   LIN {X 7.485, Y -24.478, Z 79.900}
   LaserEnd_Ext()
   LIN {X 6.429, Y -25.478, Z 79.900}
   LaserStart_Ext()
   LIN {X -3.413, Y -25.478, Z 79.900}
   LaserEnd_Ext()
   LIN {X -1.645, Y -26.478, Z 79.900}
   LaserStart_Ext()
   LIN {X 4.818, Y -26.478, Z 79.900}
   LaserEnd_Ext()
   LIN {X 0.768, Y -14.331, Z 80.750}
   LaserStart_Ext()
   LIN {X 0.932, Y -14.309, Z 80.750} C_DIS
   LIN {X 2.973, Y -14.407, Z 80.750} C_DIS
   LIN {X 4.364, Y -15.140, Z 80.750} C_DIS
   LIN {X 4.854, Y -15.396, Z 80.750} C_DIS
   LIN {X 5.246, Y -15.948, Z 80.750} C_DIS
   LIN {X 6.320, Y -17.473, Z 80.750} C_DIS
   LIN {X 6.562, Y -19.321, Z 80.750} C_DIS
   LIN {X 6.608, Y -19.665, Z 80.750} C_DIS
   LIN {X 6.497, Y -19.988, Z 80.750} C_DIS
   LIN {X 5.824, Y -21.931, Z 80.750} C_DIS
   LIN {X 4.592, Y -23.184, Z 80.750} C_DIS
   LIN {X 4.366, Y -23.413, Z 80.750} C_DIS
   LIN {X 3.828, Y -23.616, Z 80.750} C_DIS
   LIN {X 2.307, Y -24.195, Z 80.750} C_DIS
   LIN {X 1.339, Y -24.139, Z 80.750} C_DIS
   LIN {X 0.262, Y -24.074, Z 80.750} C_DIS
   LIN {X -1.038, Y -23.395, Z 80.750} C_DIS
   LIN {X -1.571, Y -23.119, Z 80.750} C_DIS
   LIN {X -1.885, Y -22.728, Z 80.750} C_DIS
   LIN {X -2.870, Y -21.491, Z 80.750} C_DIS
   LIN {X -3.249, Y -19.979, Z 80.750} C_DIS
   LIN {X -3.379, Y -19.468, Z 80.750} C_DIS
   LIN {X -3.052, Y -18.224, Z 80.750} C_DIS
   LIN {X -2.630, Y -16.631, Z 80.750} C_DIS
   LIN {X -2.228, Y -16.209, Z 80.750} C_DIS
   LIN {X -1.186, Y -15.114, Z 80.750} C_DIS
   LIN {X 0.768, Y -14.331, Z 80.750}
   LaserEnd_Ext()
   LIN {X -7.773, Y 38.728, Z 80.750}
   LaserStart_Ext()
   LIN {X -7.349, Y 37.718, Z 80.750} C_DIS
   LIN {X -6.620, Y 35.844, Z 80.750} C_DIS
   LIN {X -6.489, Y 35.509, Z 80.750} C_DIS
   LIN {X -6.365, Y 35.156, Z 80.750} C_DIS
   LIN {X -5.531, Y 32.760, Z 80.750} C_DIS
   LIN {X -5.439, Y 32.415, Z 80.750} C_DIS
   LIN {X -3.813, Y 26.595, Z 80.750} C_DIS
   LIN {X -3.780, Y 26.392, Z 80.750} C_DIS
   LIN {X -2.579, Y 19.576, Z 80.750} C_DIS
   LIN {X -1.969, Y 10.570, Z 80.750} C_DIS
   LIN {X -1.949, Y 8.966, Z 80.750} C_DIS
   LIN {X -2.076, Y 7.182, Z 80.750} C_DIS
   LIN {X -2.401, Y 1.921, Z 80.750} C_DIS
   LIN {X -2.488, Y 1.019, Z 80.750} C_DIS
   LIN {X -2.607, Y 0.242, Z 80.750} C_DIS
   LIN {X -2.989, Y -1.897, Z 80.750} C_DIS
   LIN {X -3.631, Y -5.562, Z 80.750} C_DIS
   LIN {X -4.628, Y -9.518, Z 80.750} C_DIS
   LIN {X -4.693, Y -9.777, Z 80.750} C_DIS
   LIN {X -4.739, Y -9.925, Z 80.750} C_DIS
   LIN {X -5.557, Y -12.604, Z 80.750} C_DIS
   LIN {X -6.774, Y -16.008, Z 80.750} C_DIS
   LIN {X -7.394, Y -19.162, Z 80.750} C_DIS
   LIN {X -6.873, Y -21.827, Z 80.750} C_DIS
   LIN {X -6.688, Y -22.804, Z 80.750} C_DIS
   LIN {X -6.215, Y -23.560, Z 80.750} C_DIS
   LIN {X -5.131, Y -25.266, Z 80.750} C_DIS
   LIN {X -3.475, Y -26.590, Z 80.750} C_DIS
   LIN {X -2.810, Y -27.127, Z 80.750} C_DIS
   LIN {X -0.160, Y -27.846, Z 80.750} C_DIS
   LIN {X 1.444, Y -28.255, Z 80.750} C_DIS
   LIN {X 2.595, Y -28.009, Z 80.750} C_DIS
   LIN {X 5.063, Y -27.544, Z 80.750} C_DIS
   LIN {X 6.110, Y -26.894, Z 80.750} C_DIS
   LIN {X 7.710, Y -25.848, Z 80.750} C_DIS
   LIN {X 8.986, Y -24.226, Z 80.750} C_DIS
   LIN {X 9.540, Y -23.493, Z 80.750} C_DIS
   LIN {X 9.721, Y -22.905, Z 80.750} C_DIS
   LIN {X 10.582, Y -20.217, Z 80.750} C_DIS
   LIN {X 10.827, Y -17.804, Z 80.750} C_DIS
   LIN {X 10.907, Y -16.970, Z 80.750} C_DIS
   LIN {X 10.952, Y -16.292, Z 80.750} C_DIS
   LIN {X 11.122, Y -14.017, Z 80.750} C_DIS
   LIN {X 11.251, Y -11.038, Z 80.750} C_DIS
   LIN {X 11.281, Y -10.215, Z 80.750} C_DIS
   LIN {X 11.280, Y -8.896, Z 80.750} C_DIS
   LIN {X 11.295, Y -5.428, Z 80.750} C_DIS
   LIN {X 11.137, Y -1.887, Z 80.750} C_DIS
   LIN {X 10.979, Y 1.103, Z 80.750} C_DIS
   LIN {X 10.377, Y 5.431, Z 80.750} C_DIS
   LIN {X 9.497, Y 12.340, Z 80.750} C_DIS
   LIN {X 8.336, Y 17.692, Z 80.750} C_DIS
   LIN {X 7.405, Y 21.631, Z 80.750} C_DIS
   LIN {X 6.860, Y 23.249, Z 80.750} C_DIS
   LIN {X 4.606, Y 30.446, Z 80.750} C_DIS
   LIN {X 3.585, Y 33.112, Z 80.750} C_DIS
   LIN {X 3.490, Y 33.339, Z 80.750} C_DIS
   LIN {X 3.345, Y 33.696, Z 80.750} C_DIS
   LIN {X 3.029, Y 34.443, Z 80.750} C_DIS
   LIN {X 1.716, Y 37.545, Z 80.750} C_DIS
   LIN {X 0.683, Y 39.779, Z 80.750} C_DIS
   LIN {X 0.324, Y 40.550, Z 80.750} C_DIS
   LIN {X 0.053, Y 41.100, Z 80.750} C_DIS
   LIN {X -0.525, Y 42.275, Z 80.750} C_DIS
   LIN {X -1.078, Y 43.355, Z 80.750} C_DIS
   LIN {X -1.313, Y 43.811, Z 80.750} C_DIS
   LIN {X -1.598, Y 44.174, Z 80.750} C_DIS
   LIN {X -2.220, Y 44.969, Z 80.750} C_DIS
   LIN {X -3.185, Y 45.502, Z 80.750} C_DIS
   LIN {X -3.743, Y 45.808, Z 80.750} C_DIS
   LIN {X -4.611, Y 45.864, Z 80.750} C_DIS
   LIN {X -5.484, Y 45.922, Z 80.750} C_DIS
   LIN {X -7.839, Y 44.631, Z 80.750} C_DIS
   LIN {X -8.320, Y 43.767, Z 80.750} C_DIS
   LIN {X -8.665, Y 43.160, Z 80.750} C_DIS
   LIN {X -8.736, Y 42.627, Z 80.750} C_DIS
   LIN {X -8.829, Y 41.756, Z 80.750} C_DIS
   LIN {X -8.594, Y 40.838, Z 80.750} C_DIS
   LIN {X -8.473, Y 40.337, Z 80.750} C_DIS
   LIN {X -8.219, Y 39.759, Z 80.750} C_DIS
   LIN {X -7.970, Y 39.192, Z 80.750} C_DIS
   LIN {X -7.773, Y 38.728, Z 80.750}
   LaserEnd_Ext()
   LIN {X -7.280, Y 40.107, Z 80.750}
   LaserStart_Ext()
   LIN {X -7.280, Y 43.580, Z 80.750}
   LaserEnd_Ext()
   LIN {X -6.280, Y 44.345, Z 80.750}
   LaserStart_Ext()
   LIN {X -6.280, Y 37.728, Z 80.750}
   LaserEnd_Ext()
   LIN {X -6.280, Y -18.671, Z 80.750}
   LaserStart_Ext()
   LIN {X -6.280, Y -19.649, Z 80.750}
   LaserEnd_Ext()
   LIN {X -5.280, Y -23.167, Z 80.750}
   LaserStart_Ext()
   LIN {X -5.280, Y -14.799, Z 80.750}
   LaserEnd_Ext()
   LIN {X -5.280, Y 35.081, Z 80.750}
   LaserStart_Ext()
   LIN {X -5.280, Y 44.894, Z 80.750}
   LaserEnd_Ext()
   LIN {X -4.280, Y 44.841, Z 80.750}
   LaserStart_Ext()
   LIN {X -4.280, Y 31.983, Z 80.750}
   LaserEnd_Ext()
   LIN {X -4.280, Y -11.845, Z 80.750}
   LaserStart_Ext()
   LIN {X -4.280, Y -18.961, Z 80.750}
   LaserEnd_Ext()
   LIN {X -4.280, Y -19.984, Z 80.750}
   LaserStart_Ext()
   LIN {X -4.280, Y -24.667, Z 80.750}
   LaserEnd_Ext()
   LIN {X -3.280, Y -25.466, Z 80.750}
   LaserStart_Ext()
   LIN {X -3.280, Y -22.582, Z 80.750}
   LaserEnd_Ext()
   LIN {X -3.280, Y -15.864, Z 80.750}
   LaserStart_Ext()
   LIN {X -3.280, Y -8.261, Z 80.750}
   LaserEnd_Ext()
   LIN {X -3.280, Y 28.402, Z 80.750}
   LaserStart_Ext()
   LIN {X -3.280, Y 44.412, Z 80.750}
   LaserEnd_Ext()
   LIN {X -2.280, Y 43.423, Z 80.750}
   LaserStart_Ext()
   LIN {X -2.280, Y 23.642, Z 80.750}
   LaserEnd_Ext()
   LIN {X -2.280, Y -3.644, Z 80.750}
   LaserStart_Ext()
   LIN {X -2.280, Y -14.813, Z 80.750}
   LaserEnd_Ext()
   LIN {X -2.280, Y -23.824, Z 80.750}
   LaserStart_Ext()
   LIN {X -2.280, Y -26.234, Z 80.750}
   LaserEnd_Ext()
   LIN {X -1.280, Y -26.506, Z 80.750}
   LaserStart_Ext()
   LIN {X -1.280, Y -24.397, Z 80.750}
   LaserEnd_Ext()
   LIN {X -1.280, Y -14.074, Z 80.750}
   LaserStart_Ext()
   LIN {X -1.280, Y 3.847, Z 80.750}
   LaserEnd_Ext()
   LIN {X -1.280, Y 15.194, Z 80.750}
   LaserStart_Ext()
   LIN {X -1.280, Y 41.544, Z 80.750}
   LaserEnd_Ext()
   LIN {X -0.280, Y 39.477, Z 80.750}
   LaserStart_Ext()
   LIN {X -0.280, Y -13.673, Z 80.750}
   LaserEnd_Ext()
   LIN {X -0.280, Y -24.919, Z 80.750}
   LaserStart_Ext()
   LIN {X -0.280, Y -26.777, Z 80.750}
   LaserEnd_Ext()
   LIN {X 0.720, Y -27.039, Z 80.750}
   LaserStart_Ext()
   LIN {X 0.720, Y -25.103, Z 80.750}
   LaserEnd_Ext()
   LIN {X 0.720, Y -13.312, Z 80.750}
   LaserStart_Ext()
   LIN {X 0.720, Y 37.317, Z 80.750}
   LaserEnd_Ext()
   LIN {X 1.720, Y 34.970, Z 80.750}
   LaserStart_Ext()
   LIN {X 1.720, Y -13.346, Z 80.750}
   LaserEnd_Ext()
   LIN {X 1.720, Y -25.163, Z 80.750}
   LaserStart_Ext()
   LIN {X 1.720, Y -27.173, Z 80.750}
   LaserEnd_Ext()
   LIN {X 2.720, Y -26.968, Z 80.750}
   LaserStart_Ext()
   LIN {X 2.720, Y -25.108, Z 80.750}
   LaserEnd_Ext()
   LIN {X 2.720, Y -13.394, Z 80.750}
   LaserStart_Ext()
   LIN {X 2.720, Y 32.574, Z 80.750}
   LaserEnd_Ext()
   LIN {X 3.720, Y 29.928, Z 80.750}
   LaserStart_Ext()
   LIN {X 3.720, Y -13.670, Z 80.750}
   LaserEnd_Ext()
   LIN {X 3.720, Y -24.727, Z 80.750}
   LaserStart_Ext()
   LIN {X 3.720, Y -26.780, Z 80.750}
   LaserEnd_Ext()
   LIN {X 4.720, Y -26.580, Z 80.750}
   LaserStart_Ext()
   LIN {X 4.720, Y -24.348, Z 80.750}
   LaserEnd_Ext()
   LIN {X 4.720, Y -14.198, Z 80.750}
   LaserStart_Ext()
   LIN {X 4.720, Y 26.736, Z 80.750}
   LaserEnd_Ext()
   LIN {X 5.720, Y 23.544, Z 80.750}
   LaserStart_Ext()
   LIN {X 5.720, Y -14.889, Z 80.750}
   LaserEnd_Ext()
   LIN {X 5.720, Y -23.463, Z 80.750}
   LaserStart_Ext()
   LIN {X 5.720, Y -25.954, Z 80.750}
   LaserEnd_Ext()
   LIN {X 6.720, Y -25.300, Z 80.750}
   LaserStart_Ext()
   LIN {X 6.720, Y -22.372, Z 80.750}
   LaserEnd_Ext()
   LIN {X 6.720, Y -16.305, Z 80.750}
   LaserStart_Ext()
   LIN {X 6.720, Y 20.180, Z 80.750}
   LaserEnd_Ext()
   LIN {X 7.720, Y 15.813, Z 80.750}
   LaserStart_Ext()
   LIN {X 7.720, Y -24.217, Z 80.750}
   LaserEnd_Ext()
   LIN {X 8.720, Y -22.757, Z 80.750}
   LaserStart_Ext()
   LIN {X 8.720, Y 10.522, Z 80.750}
   LaserEnd_Ext()
   LIN {X 9.720, Y 2.896, Z 80.750}
   LaserStart_Ext()
   LIN {X 9.720, Y -18.807, Z 80.750}
   LaserEnd_Ext()
   LIN {X -2.785, Y -21.446, Z 81.600}
   LaserStart_Ext()
   LIN {X -2.815, Y -21.328, Z 81.600} C_DIS
   LIN {X -3.299, Y -19.424, Z 81.600} C_DIS
   LIN {X -2.749, Y -17.335, Z 81.600} C_DIS
   LIN {X -2.557, Y -16.588, Z 81.600} C_DIS
   LIN {X -1.920, Y -15.913, Z 81.600} C_DIS
   LIN {X -1.109, Y -15.060, Z 81.600} C_DIS
   LIN {X -0.319, Y -14.744, Z 81.600} C_DIS
   LIN {X 0.911, Y -14.249, Z 81.600} C_DIS
   LIN {X 2.739, Y -14.334, Z 81.600} C_DIS
   LIN {X 3.041, Y -14.348, Z 81.600} C_DIS
   LIN {X 3.248, Y -14.457, Z 81.600} C_DIS
   LIN {X 4.925, Y -15.333, Z 81.600} C_DIS
   LIN {X 6.267, Y -17.224, Z 81.600} C_DIS
   LIN {X 6.396, Y -17.407, Z 81.600} C_DIS
   LIN {X 6.425, Y -17.629, Z 81.600} C_DIS
   LIN {X 6.689, Y -19.597, Z 81.600} C_DIS
   LIN {X 6.055, Y -21.446, Z 81.600} C_DIS
   LIN {X 5.909, Y -21.868, Z 81.600} C_DIS
   LIN {X 5.509, Y -22.274, Z 81.600} C_DIS
   LIN {X 4.458, Y -23.350, Z 81.600} C_DIS
   LIN {X 3.560, Y -23.696, Z 81.600} C_DIS
   LIN {X 2.399, Y -24.138, Z 81.600} C_DIS
   LIN {X 0.648, Y -24.037, Z 81.600} C_DIS
   LIN {X 0.353, Y -24.021, Z 81.600} C_DIS
   LIN {X 0.161, Y -23.922, Z 81.600} C_DIS
   LIN {X -1.482, Y -23.071, Z 81.600} C_DIS
   LIN {X -2.708, Y -21.542, Z 81.600} C_DIS
   LIN {X -2.785, Y -21.446, Z 81.600}
   LaserEnd_Ext()
   LIN {X -6.716, Y -16.014, Z 81.600}
   LaserStart_Ext()
   LIN {X -6.948, Y -17.246, Z 81.600} C_DIS
   LIN {X -7.315, Y -19.127, Z 81.600} C_DIS
   LIN {X -6.705, Y -22.243, Z 81.600} C_DIS
   LIN {X -6.600, Y -22.768, Z 81.600} C_DIS
   LIN {X -6.439, Y -23.019, Z 81.600} C_DIS
   LIN {X -5.037, Y -25.227, Z 81.600} C_DIS
   LIN {X -3.001, Y -26.854, Z 81.600} C_DIS
   LIN {X -2.712, Y -27.082, Z 81.600} C_DIS
   LIN {X -2.128, Y -27.209, Z 81.600} C_DIS
   LIN {X 1.739, Y -28.194, Z 81.600} C_DIS
   LIN {X 5.106, Y -27.475, Z 81.600} C_DIS
   LIN {X 5.297, Y -27.429, Z 81.600} C_DIS
   LIN {X 5.502, Y -27.300, Z 81.600} C_DIS
   LIN {X 7.745, Y -25.833, Z 81.600} C_DIS
   LIN {X 9.324, Y -23.826, Z 81.600} C_DIS
   LIN {X 9.582, Y -23.509, Z 81.600} C_DIS
   LIN {X 9.852, Y -22.677, Z 81.600} C_DIS
   LIN {X 10.664, Y -20.140, Z 81.600} C_DIS
   LIN {X 10.787, Y -18.934, Z 81.600} C_DIS
   LIN {X 10.982, Y -16.892, Z 81.600} C_DIS
   LIN {X 11.093, Y -15.232, Z 81.600} C_DIS
   LIN {X 11.189, Y -13.939, Z 81.600} C_DIS
   LIN {X 11.263, Y -12.246, Z 81.600} C_DIS
   LIN {X 11.340, Y -10.137, Z 81.600} C_DIS
   LIN {X 11.337, Y -6.755, Z 81.600} C_DIS
   LIN {X 11.343, Y -5.350, Z 81.600} C_DIS
   LIN {X 11.279, Y -3.915, Z 81.600} C_DIS
   LIN {X 11.010, Y 1.198, Z 81.600} C_DIS
   LIN {X 9.980, Y 8.597, Z 81.600} C_DIS
   LIN {X 9.457, Y 12.697, Z 81.600} C_DIS
   LIN {X 8.769, Y 15.872, Z 81.600} C_DIS
   LIN {X 7.400, Y 21.660, Z 81.600} C_DIS
   LIN {X 6.600, Y 24.039, Z 81.600} C_DIS
   LIN {X 4.603, Y 30.414, Z 81.600} C_DIS
   LIN {X 3.699, Y 32.775, Z 81.600} C_DIS
   LIN {X 3.615, Y 32.976, Z 81.600} C_DIS
   LIN {X 3.486, Y 33.292, Z 81.600} C_DIS
   LIN {X 3.353, Y 33.628, Z 81.600} C_DIS
   LIN {X 2.053, Y 36.685, Z 81.600} C_DIS
   LIN {X 1.723, Y 37.465, Z 81.600} C_DIS
   LIN {X 1.463, Y 38.027, Z 81.600} C_DIS
   LIN {X 0.328, Y 40.469, Z 81.600} C_DIS
   LIN {X -0.457, Y 42.060, Z 81.600} C_DIS
   LIN {X -0.509, Y 42.165, Z 81.600} C_DIS
   LIN {X -1.381, Y 43.859, Z 81.600} C_DIS
   LIN {X -2.087, Y 44.757, Z 81.600} C_DIS
   LIN {X -2.291, Y 45.015, Z 81.600} C_DIS
   LIN {X -2.683, Y 45.229, Z 81.600} C_DIS
   LIN {X -3.816, Y 45.851, Z 81.600} C_DIS
   LIN {X -4.788, Y 45.913, Z 81.600} C_DIS
   LIN {X -5.557, Y 45.960, Z 81.600} C_DIS
   LIN {X -7.899, Y 44.674, Z 81.600} C_DIS
   LIN {X -8.103, Y 44.309, Z 81.600} C_DIS
   LIN {X -8.736, Y 43.176, Z 81.600} C_DIS
   LIN {X -8.816, Y 42.344, Z 81.600} C_DIS
   LIN {X -8.886, Y 41.697, Z 81.600} C_DIS
   LIN {X -8.738, Y 41.121, Z 81.600} C_DIS
   LIN {X -8.532, Y 40.369, Z 81.600} C_DIS
   LIN {X -8.269, Y 39.774, Z 81.600} C_DIS
   LIN {X -8.027, Y 39.225, Z 81.600} C_DIS
   LIN {X -7.566, Y 38.137, Z 81.600} C_DIS
   LIN {X -7.403, Y 37.752, Z 81.600} C_DIS
   LIN {X -7.225, Y 37.303, Z 81.600} C_DIS
   LIN {X -6.537, Y 35.545, Z 81.600} C_DIS
   LIN {X -5.613, Y 32.910, Z 81.600} C_DIS
   LIN {X -5.573, Y 32.799, Z 81.600} C_DIS
   LIN {X -3.889, Y 26.817, Z 81.600} C_DIS
   LIN {X -3.656, Y 25.742, Z 81.600} C_DIS
   LIN {X -2.630, Y 19.923, Z 81.600} C_DIS
   LIN {X -1.942, Y 9.757, Z 81.600} C_DIS
   LIN {X -1.913, Y 9.438, Z 81.600} C_DIS
   LIN {X -1.913, Y 9.323, Z 81.600} C_DIS
   LIN {X -2.355, Y 2.148, Z 81.600} C_DIS
   LIN {X -2.481, Y 0.845, Z 81.600} C_DIS
   LIN {X -2.653, Y -0.278, Z 81.600} C_DIS
   LIN {X -3.206, Y -3.370, Z 81.600} C_DIS
   LIN {X -3.577, Y -5.490, Z 81.600} C_DIS
   LIN {X -4.234, Y -8.099, Z 81.600} C_DIS
   LIN {X -4.637, Y -9.740, Z 81.600} C_DIS
   LIN {X -4.984, Y -10.889, Z 81.600} C_DIS
   LIN {X -5.530, Y -12.677, Z 81.600} C_DIS
   LIN {X -6.260, Y -14.720, Z 81.600} C_DIS
   LIN {X -6.716, Y -16.014, Z 81.600}
   LaserEnd_Ext()
   LIN {X 5.112, Y -26.360, Z 81.600}
   LaserStart_Ext()
   LIN {X -1.409, Y -26.360, Z 81.600}
   LaserEnd_Ext()
   LIN {X -3.268, Y -25.360, Z 81.600}
   LaserStart_Ext()
   LIN {X 6.641, Y -25.360, Z 81.600}
   LaserEnd_Ext()
   LIN {X 7.632, Y -24.360, Z 81.600}
   LaserStart_Ext()
   LIN {X 4.617, Y -24.360, Z 81.600}
   LaserEnd_Ext()
   LIN {X -1.168, Y -24.360, Z 81.600}
   LaserStart_Ext()
   LIN {X -4.403, Y -24.360, Z 81.600}
   LaserEnd_Ext()
   LIN {X -5.038, Y -23.360, Z 81.600}
   LaserStart_Ext()
   LIN {X -2.532, Y -23.360, Z 81.600}
   LaserEnd_Ext()
   LIN {X 5.846, Y -23.360, Z 81.600}
   LaserStart_Ext()
   LIN {X 8.418, Y -23.360, Z 81.600}
   LaserEnd_Ext()
   LIN {X 8.903, Y -22.360, Z 81.600}
   LaserStart_Ext()
   LIN {X 6.779, Y -22.360, Z 81.600}
   LaserEnd_Ext()
   LIN {X -3.334, Y -22.360, Z 81.600}
   LaserStart_Ext()
   LIN {X -5.662, Y -22.360, Z 81.600}
   LaserEnd_Ext()
   LIN {X -5.859, Y -21.360, Z 81.600}
   LaserStart_Ext()
   LIN {X -3.838, Y -21.360, Z 81.600}
   LaserEnd_Ext()
   LIN {X 7.142, Y -21.360, Z 81.600}
   LaserStart_Ext()
   LIN {X 9.224, Y -21.360, Z 81.600}
   LaserEnd_Ext()
   LIN {X 9.544, Y -20.360, Z 81.600}
   LaserStart_Ext()
   LIN {X 7.485, Y -20.360, Z 81.600}
   LaserEnd_Ext()
   LIN {X -4.093, Y -20.360, Z 81.600}
   LaserStart_Ext()
   LIN {X -6.055, Y -20.360, Z 81.600}
   LaserEnd_Ext()
   LIN {X -6.250, Y -19.360, Z 81.600}
   LaserStart_Ext()
   LIN {X -4.297, Y -19.360, Z 81.600}
   LaserEnd_Ext()
   LIN {X 7.666, Y -19.360, Z 81.600}
   LaserStart_Ext()
   LIN {X 9.739, Y -19.360, Z 81.600}
   LaserEnd_Ext()
   LIN {X 9.837, Y -18.360, Z 81.600}
   LaserStart_Ext()
   LIN {X 7.532, Y -18.360, Z 81.600}
   LaserEnd_Ext()
   LIN {X -4.053, Y -18.360, Z 81.600}
   LaserStart_Ext()
   LIN {X -6.146, Y -18.360, Z 81.600}
   LaserEnd_Ext()
   LIN {X -5.952, Y -17.360, Z 81.600}
   LaserStart_Ext()
   LIN {X -3.789, Y -17.360, Z 81.600}
   LaserEnd_Ext()
   LIN {X 7.398, Y -17.360, Z 81.600}
   LaserStart_Ext()
   LIN {X 9.933, Y -17.360, Z 81.600}
   LaserEnd_Ext()
   LIN {X 10.015, Y -16.360, Z 81.600}
   LaserStart_Ext()
   LIN {X 6.880, Y -16.360, Z 81.600}
   LaserEnd_Ext()
   LIN {X -3.531, Y -16.360, Z 81.600}
   LaserStart_Ext()
   LIN {X -5.764, Y -16.360, Z 81.600}
   LaserEnd_Ext()
   LIN {X -5.425, Y -15.360, Z 81.600}
   LaserStart_Ext()
   LIN {X -2.773, Y -15.360, Z 81.600}
   LaserEnd_Ext()
   LIN {X 6.170, Y -15.360, Z 81.600}
   LaserStart_Ext()
   LIN {X 10.082, Y -15.360, Z 81.600}
   LaserEnd_Ext()
   LIN {X 10.155, Y -14.360, Z 81.600}
   LaserStart_Ext()
   LIN {X 5.222, Y -14.360, Z 81.600}
   LaserEnd_Ext()
   LIN {X -1.822, Y -14.360, Z 81.600}
   LaserStart_Ext()
   LIN {X -5.070, Y -14.360, Z 81.600}
   LaserEnd_Ext()
   LIN {X -4.712, Y -13.360, Z 81.600}
   LaserStart_Ext()
   LIN {X 0.441, Y -13.360, Z 81.600}
   LaserEnd_Ext()
   LIN {X 3.193, Y -13.360, Z 81.600}
   LaserStart_Ext()
   LIN {X 10.214, Y -13.360, Z 81.600}
   LaserEnd_Ext()
   LIN {X 10.257, Y -12.360, Z 81.600}
   LaserStart_Ext()
   LIN {X -4.388, Y -12.360, Z 81.600}
   LaserEnd_Ext()
   LIN {X -4.082, Y -11.360, Z 81.600}
   LaserStart_Ext()
   LIN {X 10.295, Y -11.360, Z 81.600}
   LaserEnd_Ext()
   LIN {X 10.331, Y -10.360, Z 81.600}
   LaserStart_Ext()
   LIN {X -3.779, Y -10.360, Z 81.600}
   LaserEnd_Ext()
   LIN {X -3.514, Y -9.360, Z 81.600}
   LaserStart_Ext()
   LIN {X 10.339, Y -9.360, Z 81.600}
   LaserEnd_Ext()
   LIN {X 10.338, Y -8.360, Z 81.600}
   LaserStart_Ext()
   LIN {X -3.269, Y -8.360, Z 81.600}
   LaserEnd_Ext()
   LIN {X -3.017, Y -7.360, Z 81.600}
   LaserStart_Ext()
   LIN {X 10.337, Y -7.360, Z 81.600}
   LaserEnd_Ext()
   LIN {X 10.338, Y -6.360, Z 81.600}
   LaserStart_Ext()
   LIN {X -2.765, Y -6.360, Z 81.600}
   LaserEnd_Ext()
   LIN {X -2.539, Y -5.360, Z 81.600}
   LaserStart_Ext()
   LIN {X 10.342, Y -5.360, Z 81.600}
   LaserEnd_Ext()
   LIN {X 10.298, Y -4.360, Z 81.600}
   LaserStart_Ext()
   LIN {X -2.364, Y -4.360, Z 81.600}
   LaserEnd_Ext()
   LIN {X -2.188, Y -3.360, Z 81.600}
   LaserStart_Ext()
   LIN {X 10.248, Y -3.360, Z 81.600}
   LaserEnd_Ext()
   LIN {X 10.196, Y -2.360, Z 81.600}
   LaserStart_Ext()
   LIN {X -2.009, Y -2.360, Z 81.600}
   LaserEnd_Ext()
   LIN {X -1.831, Y -1.360, Z 81.600}
   LaserStart_Ext()
   LIN {X 10.143, Y -1.360, Z 81.600}
   LaserEnd_Ext()
   LIN {X 10.090, Y -0.360, Z 81.600}
   LaserStart_Ext()
   LIN {X -1.654, Y -0.360, Z 81.600}
   LaserEnd_Ext()
   LIN {X -1.501, Y 0.640, Z 81.600}
   LaserStart_Ext()
   LIN {X 10.038, Y 0.640, Z 81.600}
   LaserEnd_Ext()
   LIN {X 9.939, Y 1.640, Z 81.600}
   LaserStart_Ext()
   LIN {X -1.400, Y 1.640, Z 81.600}
   LaserEnd_Ext()
   LIN {X -1.323, Y 2.640, Z 81.600}
   LaserStart_Ext()
   LIN {X 9.800, Y 2.640, Z 81.600}
   LaserEnd_Ext()
   LIN {X 9.660, Y 3.640, Z 81.600}
   LaserStart_Ext()
   LIN {X -1.261, Y 3.640, Z 81.600}
   LaserEnd_Ext()
   LIN {X -1.200, Y 4.640, Z 81.600}
   LaserStart_Ext()
   LIN {X 9.521, Y 4.640, Z 81.600}
   LaserEnd_Ext()
   LIN {X 9.382, Y 5.640, Z 81.600}
   LaserStart_Ext()
   LIN {X -1.138, Y 5.640, Z 81.600}
   LaserEnd_Ext()
   LIN {X -1.076, Y 6.640, Z 81.600}
   LaserStart_Ext()
   LIN {X 9.243, Y 6.640, Z 81.600}
   LaserEnd_Ext()
   LIN {X 9.103, Y 7.640, Z 81.600}
   LaserStart_Ext()
   LIN {X -1.015, Y 7.640, Z 81.600}
   LaserEnd_Ext()
   LIN {X -0.953, Y 8.640, Z 81.600}
   LaserStart_Ext()
   LIN {X 8.966, Y 8.640, Z 81.600}
   LaserEnd_Ext()
   LIN {X 8.839, Y 9.640, Z 81.600}
   LaserStart_Ext()
   LIN {X -0.927, Y 9.640, Z 81.600}
   LaserEnd_Ext()
   LIN {X -1.000, Y 10.640, Z 81.600}
   LaserStart_Ext()
   LIN {X 8.711, Y 10.640, Z 81.600}
   LaserEnd_Ext()
   LIN {X 8.584, Y 11.640, Z 81.600}
   LaserStart_Ext()
   LIN {X -1.067, Y 11.640, Z 81.600}
   LaserEnd_Ext()
   LIN {X -1.135, Y 12.640, Z 81.600}
   LaserStart_Ext()
   LIN {X 8.447, Y 12.640, Z 81.600}
   LaserEnd_Ext()
   LIN {X 8.230, Y 13.640, Z 81.600}
   LaserStart_Ext()
   LIN {X -1.202, Y 13.640, Z 81.600}
   LaserEnd_Ext()
   LIN {X -1.270, Y 14.640, Z 81.600}
   LaserStart_Ext()
   LIN {X 8.013, Y 14.640, Z 81.600}
   LaserEnd_Ext()
   LIN {X 7.796, Y 15.640, Z 81.600}
   LaserStart_Ext()
   LIN {X -1.338, Y 15.640, Z 81.600}
   LaserEnd_Ext()
   LIN {X -1.405, Y 16.640, Z 81.600}
   LaserStart_Ext()
   LIN {X 7.560, Y 16.640, Z 81.600}
   LaserEnd_Ext()
   LIN {X 7.323, Y 17.640, Z 81.600}
   LaserStart_Ext()
   LIN {X -1.473, Y 17.640, Z 81.600}
   LaserEnd_Ext()
   LIN {X -1.541, Y 18.640, Z 81.600}
   LaserStart_Ext()
   LIN {X 7.087, Y 18.640, Z 81.600}
   LaserEnd_Ext()
   LIN {X 6.850, Y 19.640, Z 81.600}
   LaserStart_Ext()
   LIN {X -1.608, Y 19.640, Z 81.600}
   LaserEnd_Ext()
   LIN {X -1.741, Y 20.640, Z 81.600}
   LaserStart_Ext()
   LIN {X 6.614, Y 20.640, Z 81.600}
   LaserEnd_Ext()
   LIN {X 6.352, Y 21.640, Z 81.600}
   LaserStart_Ext()
   LIN {X -1.917, Y 21.640, Z 81.600}
   LaserEnd_Ext()
   LIN {X -2.093, Y 22.640, Z 81.600}
   LaserStart_Ext()
   LIN {X 6.016, Y 22.640, Z 81.600}
   LaserEnd_Ext()
   LIN {X 5.679, Y 23.640, Z 81.600}
   LaserStart_Ext()
   LIN {X -2.270, Y 23.640, Z 81.600}
   LaserEnd_Ext()
   LIN {X -2.446, Y 24.640, Z 81.600}
   LaserStart_Ext()
   LIN {X 5.364, Y 24.640, Z 81.600}
   LaserEnd_Ext()
   LIN {X 5.051, Y 25.640, Z 81.600}
   LaserStart_Ext()
   LIN {X -2.622, Y 25.640, Z 81.600}
   LaserEnd_Ext()
   LIN {X -2.828, Y 26.640, Z 81.600}
   LaserStart_Ext()
   LIN {X 4.738, Y 26.640, Z 81.600}
   LaserEnd_Ext()
   LIN {X 4.424, Y 27.640, Z 81.600}
   LaserStart_Ext()
   LIN {X -3.082, Y 27.640, Z 81.600}
   LaserEnd_Ext()
   LIN {X -3.364, Y 28.640, Z 81.600}
   LaserStart_Ext()
   LIN {X 4.111, Y 28.640, Z 81.600}
   LaserEnd_Ext()
   LIN {X 3.798, Y 29.640, Z 81.600}
   LaserStart_Ext()
   LIN {X -3.645, Y 29.640, Z 81.600}
   LaserEnd_Ext()
   LIN {X -3.926, Y 30.640, Z 81.600}
   LaserStart_Ext()
   LIN {X 3.446, Y 30.640, Z 81.600}
   LaserEnd_Ext()
   LIN {X 3.063, Y 31.640, Z 81.600}
   LaserStart_Ext()
   LIN {X -4.208, Y 31.640, Z 81.600}
   LaserEnd_Ext()
   LIN {X -4.489, Y 32.640, Z 81.600}
   LaserStart_Ext()
   LIN {X 2.672, Y 32.640, Z 81.600}
   LaserEnd_Ext()
   LIN {X 2.261, Y 33.640, Z 81.600}
   LaserStart_Ext()
   LIN {X -4.809, Y 33.640, Z 81.600}
   LaserEnd_Ext()
   LIN {X -5.160, Y 34.640, Z 81.600}
   LaserStart_Ext()
   LIN {X 1.836, Y 34.640, Z 81.600}
   LaserEnd_Ext()
   LIN {X 1.411, Y 35.640, Z 81.600}
   LaserStart_Ext()
   LIN {X -5.511, Y 35.640, Z 81.600}
   LaserEnd_Ext()
   LIN {X -5.892, Y 36.640, Z 81.600}
   LaserStart_Ext()
   LIN {X 0.987, Y 36.640, Z 81.600}
   LaserEnd_Ext()
   LIN {X 0.540, Y 37.640, Z 81.600}
   LaserStart_Ext()
   LIN {X -6.284, Y 37.640, Z 81.600}
   LaserEnd_Ext()
   LIN {X -6.693, Y 38.640, Z 81.600}
   LaserStart_Ext()
   LIN {X 0.076, Y 38.640, Z 81.600}
   LaserEnd_Ext()
   LIN {X -0.389, Y 39.640, Z 81.600}
   LaserStart_Ext()
   LIN {X -7.117, Y 39.640, Z 81.600}
   LaserEnd_Ext()
   LIN {X -7.559, Y 40.640, Z 81.600}
   LaserStart_Ext()
   LIN {X -0.871, Y 40.640, Z 81.600}
   LaserEnd_Ext()
   LIN {X -1.365, Y 41.640, Z 81.600}
   LaserStart_Ext()
   LIN {X -7.839, Y 41.640, Z 81.600}
   LaserEnd_Ext()
   LIN {X -7.783, Y 42.640, Z 81.600}
   LaserStart_Ext()
   LIN {X -1.878, Y 42.640, Z 81.600}
   LaserEnd_Ext()
   LIN {X -2.480, Y 43.640, Z 81.600}
   LaserStart_Ext()
   LIN {X -7.331, Y 43.640, Z 81.600}
   LaserEnd_Ext()
   LIN {X -5.884, Y 44.640, Z 81.600}
   LaserStart_Ext()
   LIN {X -3.688, Y 44.640, Z 81.600}
   LaserEnd_Ext()
   LIN {X -3.044, Y -20.068, Z 82.450}
   LaserStart_Ext()
   LIN {X -3.219, Y -19.380, Z 82.450} C_DIS
   LIN {X -3.042, Y -18.710, Z 82.450} C_DIS
   LIN {X -2.490, Y -16.552, Z 82.450} C_DIS
   LIN {X -1.313, Y -15.306, Z 82.450} C_DIS
   LIN {X -1.047, Y -15.017, Z 82.450} C_DIS
   LIN {X -0.475, Y -14.782, Z 82.450} C_DIS
   LIN {X 0.987, Y -14.194, Z 82.450} C_DIS
   LIN {X 2.062, Y -14.244, Z 82.450} C_DIS
   LIN {X 3.110, Y -14.289, Z 82.450} C_DIS
   LIN {X 4.242, Y -14.876, Z 82.450} C_DIS
   LIN {X 4.995, Y -15.270, Z 82.450} C_DIS
   LIN {X 5.569, Y -16.077, Z 82.450} C_DIS
   LIN {X 6.472, Y -17.340, Z 82.450} C_DIS
   LIN {X 6.647, Y -18.614, Z 82.450} C_DIS
   LIN {X 6.770, Y -19.530, Z 82.450} C_DIS
   LIN {X 6.410, Y -20.579, Z 82.450} C_DIS
   LIN {X 6.012, Y -21.775, Z 82.450} C_DIS
   LIN {X 5.381, Y -22.437, Z 82.450} C_DIS
   LIN {X 4.551, Y -23.285, Z 82.450} C_DIS
   LIN {X 2.592, Y -24.041, Z 82.450} C_DIS
   LIN {X 2.491, Y -24.080, Z 82.450} C_DIS
   LIN {X 0.444, Y -23.969, Z 82.450} C_DIS
   LIN {X -0.955, Y -23.250, Z 82.450} C_DIS
   LIN {X -1.393, Y -23.023, Z 82.450} C_DIS
   LIN {X -1.764, Y -22.561, Z 82.450} C_DIS
   LIN {X -2.700, Y -21.401, Z 82.450} C_DIS
   LIN {X -3.044, Y -20.068, Z 82.450}
   LaserEnd_Ext()
   LIN {X 11.056, Y -16.815, Z 82.450}
   LaserStart_Ext()
   LIN {X 11.234, Y -14.172, Z 82.450} C_DIS
   LIN {X 11.257, Y -13.861, Z 82.450} C_DIS
   LIN {X 11.275, Y -13.454, Z 82.450} C_DIS
   LIN {X 11.399, Y -10.058, Z 82.450} C_DIS
   LIN {X 11.395, Y -5.797, Z 82.450} C_DIS
   LIN {X 11.391, Y -5.271, Z 82.450} C_DIS
   LIN {X 11.376, Y -5.087, Z 82.450} C_DIS
   LIN {X 11.041, Y 1.292, Z 82.450} C_DIS
   LIN {X 9.583, Y 11.764, Z 82.450} C_DIS
   LIN {X 9.418, Y 13.054, Z 82.450} C_DIS
   LIN {X 9.202, Y 14.053, Z 82.450} C_DIS
   LIN {X 7.396, Y 21.690, Z 82.450} C_DIS
   LIN {X 6.340, Y 24.828, Z 82.450} C_DIS
   LIN {X 4.601, Y 30.381, Z 82.450} C_DIS
   LIN {X 3.813, Y 32.438, Z 82.450} C_DIS
   LIN {X 3.740, Y 32.613, Z 82.450} C_DIS
   LIN {X 3.628, Y 32.889, Z 82.450} C_DIS
   LIN {X 3.391, Y 33.487, Z 82.450} C_DIS
   LIN {X 2.033, Y 36.681, Z 82.450} C_DIS
   LIN {X 1.691, Y 37.473, Z 82.450} C_DIS
   LIN {X 0.373, Y 40.302, Z 82.450} C_DIS
   LIN {X 0.265, Y 40.521, Z 82.450} C_DIS
   LIN {X -0.666, Y 42.396, Z 82.450} C_DIS
   LIN {X -1.364, Y 43.746, Z 82.450} C_DIS
   LIN {X -1.449, Y 43.907, Z 82.450} C_DIS
   LIN {X -1.579, Y 44.072, Z 82.450} C_DIS
   LIN {X -2.362, Y 45.060, Z 82.450} C_DIS
   LIN {X -3.513, Y 45.689, Z 82.450} C_DIS
   LIN {X -3.889, Y 45.893, Z 82.450} C_DIS
   LIN {X -4.715, Y 45.942, Z 82.450} C_DIS
   LIN {X -5.630, Y 45.998, Z 82.450} C_DIS
   LIN {X -6.290, Y 45.636, Z 82.450} C_DIS
   LIN {X -7.981, Y 44.692, Z 82.450} C_DIS
   LIN {X -8.592, Y 43.589, Z 82.450} C_DIS
   LIN {X -8.798, Y 43.220, Z 82.450} C_DIS
   LIN {X -8.846, Y 42.721, Z 82.450} C_DIS
   LIN {X -8.949, Y 41.722, Z 82.450} C_DIS
   LIN {X -8.720, Y 40.868, Z 82.450} C_DIS
   LIN {X -8.592, Y 40.400, Z 82.450} C_DIS
   LIN {X -8.374, Y 39.909, Z 82.450} C_DIS
   LIN {X -8.084, Y 39.257, Z 82.450} C_DIS
   LIN {X -7.855, Y 38.723, Z 82.450} C_DIS
   LIN {X -7.456, Y 37.786, Z 82.450} C_DIS
   LIN {X -6.772, Y 36.049, Z 82.450} C_DIS
   LIN {X -6.586, Y 35.581, Z 82.450} C_DIS
   LIN {X -6.429, Y 35.143, Z 82.450} C_DIS
   LIN {X -5.615, Y 32.837, Z 82.450} C_DIS
   LIN {X -5.409, Y 32.177, Z 82.450} C_DIS
   LIN {X -3.977, Y 27.086, Z 82.450} C_DIS
   LIN {X -3.479, Y 24.799, Z 82.450} C_DIS
   LIN {X -2.681, Y 20.270, Z 82.450} C_DIS
   LIN {X -2.146, Y 12.358, Z 82.450} C_DIS
   LIN {X -1.912, Y 9.787, Z 82.450} C_DIS
   LIN {X -1.910, Y 8.861, Z 82.450} C_DIS
   LIN {X -2.310, Y 2.375, Z 82.450} C_DIS
   LIN {X -2.475, Y 0.671, Z 82.450} C_DIS
   LIN {X -2.700, Y -0.798, Z 82.450} C_DIS
   LIN {X -3.422, Y -4.842, Z 82.450} C_DIS
   LIN {X -3.523, Y -5.418, Z 82.450} C_DIS
   LIN {X -3.702, Y -6.126, Z 82.450} C_DIS
   LIN {X -4.571, Y -9.670, Z 82.450} C_DIS
   LIN {X -5.320, Y -12.152, Z 82.450} C_DIS
   LIN {X -5.503, Y -12.750, Z 82.450} C_DIS
   LIN {X -5.746, Y -13.432, Z 82.450} C_DIS
   LIN {X -6.643, Y -15.978, Z 82.450} C_DIS
   LIN {X -7.101, Y -18.403, Z 82.450} C_DIS
   LIN {X -7.235, Y -19.093, Z 82.450} C_DIS
   LIN {X -7.012, Y -20.236, Z 82.450} C_DIS
   LIN {X -6.511, Y -22.732, Z 82.450} C_DIS
   LIN {X -5.748, Y -23.920, Z 82.450} C_DIS
   LIN {X -4.943, Y -25.187, Z 82.450} C_DIS
   LIN {X -3.775, Y -26.121, Z 82.450} C_DIS
   LIN {X -2.613, Y -27.036, Z 82.450} C_DIS
   LIN {X -0.265, Y -27.547, Z 82.450} C_DIS
   LIN {X 2.035, Y -28.133, Z 82.450} C_DIS
   LIN {X 4.036, Y -27.706, Z 82.450} C_DIS
   LIN {X 5.309, Y -27.402, Z 82.450} C_DIS
   LIN {X 6.677, Y -26.540, Z 82.450} C_DIS
   LIN {X 7.780, Y -25.818, Z 82.450} C_DIS
   LIN {X 8.557, Y -24.831, Z 82.450} C_DIS
   LIN {X 9.626, Y -23.515, Z 82.450} C_DIS
   LIN {X 10.747, Y -20.064, Z 82.450} C_DIS
   LIN {X 11.056, Y -16.815, Z 82.450}
   LaserEnd_Ext()
   LIN {X 9.602, Y -20.352, Z 82.450}
   LaserStart_Ext()
   LIN {X 9.602, Y 4.373, Z 82.450}
   LaserEnd_Ext()
   LIN {X 8.602, Y 11.556, Z 82.450}
   LaserStart_Ext()
   LIN {X 8.602, Y -23.190, Z 82.450}
   LaserEnd_Ext()
   LIN {X 7.602, Y -24.428, Z 82.450}
   LaserStart_Ext()
   LIN {X 7.602, Y -20.187, Z 82.450}
   LaserEnd_Ext()
   LIN {X 7.602, Y -18.218, Z 82.450}
   LaserStart_Ext()
   LIN {X 7.602, Y 16.472, Z 82.450}
   LaserEnd_Ext()
   LIN {X 6.602, Y 20.702, Z 82.450}
   LaserStart_Ext()
   LIN {X 6.602, Y -15.803, Z 82.450}
   LaserEnd_Ext()
   LIN {X 6.602, Y -22.605, Z 82.450}
   LaserStart_Ext()
   LIN {X 6.602, Y -25.394, Z 82.450}
   LaserEnd_Ext()
   LIN {X 5.602, Y -26.035, Z 82.450}
   LaserStart_Ext()
   LIN {X 5.602, Y -23.641, Z 82.450}
   LaserEnd_Ext()
   LIN {X 5.602, Y -14.475, Z 82.450}
   LaserStart_Ext()
   LIN {X 5.602, Y 23.887, Z 82.450}
   LaserEnd_Ext()
   LIN {X 4.602, Y 27.033, Z 82.450}
   LaserStart_Ext()
   LIN {X 4.602, Y -13.936, Z 82.450}
   LaserEnd_Ext()
   LIN {X 4.602, Y -24.337, Z 82.450}
   LaserStart_Ext()
   LIN {X 4.602, Y -26.543, Z 82.450}
   LaserEnd_Ext()
   LIN {X 3.602, Y -26.776, Z 82.450}
   LaserStart_Ext()
   LIN {X 3.602, Y -24.723, Z 82.450}
   LaserEnd_Ext()
   LIN {X 3.602, Y -13.418, Z 82.450}
   LaserStart_Ext()
   LIN {X 3.602, Y 30.194, Z 82.450}
   LaserEnd_Ext()
   LIN {X 2.602, Y 32.763, Z 82.450}
   LaserStart_Ext()
   LIN {X 2.602, Y -13.266, Z 82.450}
   LaserEnd_Ext()
   LIN {X 2.602, Y -25.073, Z 82.450}
   LaserStart_Ext()
   LIN {X 2.602, Y -26.990, Z 82.450}
   LaserEnd_Ext()
   LIN {X 1.602, Y -26.991, Z 82.450}
   LaserStart_Ext()
   LIN {X 1.602, Y -25.034, Z 82.450}
   LaserEnd_Ext()
   LIN {X 1.602, Y -13.221, Z 82.450}
   LaserStart_Ext()
   LIN {X 1.602, Y 35.138, Z 82.450}
   LaserEnd_Ext()
   LIN {X 0.602, Y 37.443, Z 82.450}
   LaserStart_Ext()
   LIN {X 0.602, Y -13.271, Z 82.450}
   LaserEnd_Ext()
   LIN {X 0.602, Y -24.979, Z 82.450}
   LaserStart_Ext()
   LIN {X 0.602, Y -26.736, Z 82.450}
   LaserEnd_Ext()
   LIN {X -0.398, Y -26.495, Z 82.450}
   LaserStart_Ext()
   LIN {X -0.398, Y -24.660, Z 82.450}
   LaserEnd_Ext()
   LIN {X -0.398, Y -13.673, Z 82.450}
   LaserStart_Ext()
   LIN {X -0.398, Y 39.588, Z 82.450}
   LaserEnd_Ext()
   LIN {X -1.398, Y 41.623, Z 82.450}
   LaserStart_Ext()
   LIN {X -1.398, Y 16.119, Z 82.450}
   LaserEnd_Ext()
   LIN {X -1.398, Y 1.419, Z 82.450}
   LaserStart_Ext()
   LIN {X -1.398, Y -14.080, Z 82.450}
   LaserEnd_Ext()
   LIN {X -1.398, Y -24.146, Z 82.450}
   LaserStart_Ext()
   LIN {X -1.398, Y -26.277, Z 82.450}
   LaserEnd_Ext()
   LIN {X -2.398, Y -25.933, Z 82.450}
   LaserStart_Ext()
   LIN {X -2.398, Y -23.368, Z 82.450}
   LaserEnd_Ext()
   LIN {X -2.398, Y -14.999, Z 82.450}
   LaserStart_Ext()
   LIN {X -2.398, Y -4.795, Z 82.450}
   LaserEnd_Ext()
   LIN {X -2.398, Y 24.424, Z 82.450}
   LaserStart_Ext()
   LIN {X -2.398, Y 43.495, Z 82.450}
   LaserEnd_Ext()
   LIN {X -3.398, Y 44.487, Z 82.450}
   LaserStart_Ext()
   LIN {X -3.398, Y 28.720, Z 82.450}
   LaserEnd_Ext()
   LIN {X -3.398, Y -9.086, Z 82.450}
   LaserStart_Ext()
   LIN {X -3.398, Y -16.136, Z 82.450}
   LaserEnd_Ext()
   LIN {X -3.398, Y -22.128, Z 82.450}
   LaserStart_Ext()
   LIN {X -3.398, Y -25.142, Z 82.450}
   LaserEnd_Ext()
   LIN {X -4.398, Y -24.180, Z 82.450}
   LaserStart_Ext()
   LIN {X -4.398, Y -12.557, Z 82.450}
   LaserEnd_Ext()
   LIN {X -4.398, Y 32.274, Z 82.450}
   LaserStart_Ext()
   LIN {X -4.398, Y 44.922, Z 82.450}
   LaserEnd_Ext()
   LIN {X -5.398, Y 44.982, Z 82.450}
   LaserStart_Ext()
   LIN {X -5.398, Y 35.225, Z 82.450}
   LaserEnd_Ext()
   LIN {X -5.398, Y -15.453, Z 82.450}
   LaserStart_Ext()
   LIN {X -5.398, Y -22.615, Z 82.450}
   LaserEnd_Ext()
   LIN {X -6.398, Y 37.828, Z 82.450}
   LaserStart_Ext()
   LIN {X -6.398, Y 44.430, Z 82.450}
   LaserEnd_Ext()
   LIN {X -7.398, Y 43.681, Z 82.450}
   LaserStart_Ext()
   LIN {X -7.398, Y 40.175, Z 82.450}
   LaserEnd_Ext()
   LIN {X -3.138, Y -19.336, Z 83.300}
   LaserStart_Ext()
   LIN {X -2.716, Y -17.663, Z 83.300} C_DIS
   LIN {X -2.422, Y -16.516, Z 83.300} C_DIS
   LIN {X -2.110, Y -16.186, Z 83.300} C_DIS
   LIN {X -1.014, Y -14.995, Z 83.300} C_DIS
   LIN {X 0.866, Y -14.222, Z 83.300} C_DIS
   LIN {X 1.063, Y -14.139, Z 83.300} C_DIS
   LIN {X 1.319, Y -14.150, Z 83.300} C_DIS
   LIN {X 3.179, Y -14.230, Z 83.300} C_DIS
   LIN {X 4.531, Y -14.932, Z 83.300} C_DIS
   LIN {X 5.066, Y -15.206, Z 83.300} C_DIS
   LIN {X 5.537, Y -15.860, Z 83.300} C_DIS
   LIN {X 6.548, Y -17.273, Z 83.300} C_DIS
   LIN {X 6.764, Y -18.847, Z 83.300} C_DIS
   LIN {X 6.851, Y -19.462, Z 83.300} C_DIS
   LIN {X 6.661, Y -20.051, Z 83.300} C_DIS
   LIN {X 6.123, Y -21.670, Z 83.300} C_DIS
   LIN {X 4.691, Y -23.171, Z 83.300} C_DIS
   LIN {X 4.607, Y -23.235, Z 83.300} C_DIS
   LIN {X 2.593, Y -24.021, Z 83.300} C_DIS
   LIN {X 1.236, Y -23.954, Z 83.300} C_DIS
   LIN {X 0.536, Y -23.916, Z 83.300} C_DIS
   LIN {X -0.314, Y -23.480, Z 83.300} C_DIS
   LIN {X -1.304, Y -22.974, Z 83.300} C_DIS
   LIN {X -1.840, Y -22.315, Z 83.300} C_DIS
   LIN {X -2.615, Y -21.356, Z 83.300} C_DIS
   LIN {X -2.946, Y -20.071, Z 83.300} C_DIS
   LIN {X -3.138, Y -19.336, Z 83.300}
   LaserEnd_Ext()
   LIN {X -5.703, Y 46.036, Z 83.300}
   LaserStart_Ext()
   LIN {X -7.467, Y 45.040, Z 83.300} C_DIS
   LIN {X -8.069, Y 44.704, Z 83.300} C_DIS
   LIN {X -8.264, Y 44.352, Z 83.300} C_DIS
   LIN {X -8.860, Y 43.265, Z 83.300} C_DIS
   LIN {X -8.989, Y 42.091, Z 83.300} C_DIS
   LIN {X -9.017, Y 41.816, Z 83.300} C_DIS
   LIN {X -8.947, Y 41.554, Z 83.300} C_DIS
   LIN {X -8.652, Y 40.431, Z 83.300} C_DIS
   LIN {X -8.362, Y 39.784, Z 83.300} C_DIS
   LIN {X -8.141, Y 39.289, Z 83.300} C_DIS
   LIN {X -7.721, Y 38.309, Z 83.300} C_DIS
   LIN {X -7.510, Y 37.819, Z 83.300} C_DIS
   LIN {X -7.309, Y 37.317, Z 83.300} C_DIS
   LIN {X -6.634, Y 35.617, Z 83.300} C_DIS
   LIN {X -5.694, Y 32.979, Z 83.300} C_DIS
   LIN {X -5.657, Y 32.875, Z 83.300} C_DIS
   LIN {X -5.252, Y 31.576, Z 83.300} C_DIS
   LIN {X -4.064, Y 27.355, Z 83.300} C_DIS
   LIN {X -3.303, Y 23.856, Z 83.300} C_DIS
   LIN {X -2.732, Y 20.617, Z 83.300} C_DIS
   LIN {X -2.350, Y 14.959, Z 83.300} C_DIS
   LIN {X -1.911, Y 10.136, Z 83.300} C_DIS
   LIN {X -1.908, Y 8.398, Z 83.300} C_DIS
   LIN {X -2.265, Y 2.602, Z 83.300} C_DIS
   LIN {X -2.469, Y 0.497, Z 83.300} C_DIS
   LIN {X -2.746, Y -1.318, Z 83.300} C_DIS
   LIN {X -3.392, Y -4.932, Z 83.300} C_DIS
   LIN {X -3.496, Y -5.473, Z 83.300} C_DIS
   LIN {X -3.789, Y -6.681, Z 83.300} C_DIS
   LIN {X -4.505, Y -9.601, Z 83.300} C_DIS
   LIN {X -5.203, Y -11.913, Z 83.300} C_DIS
   LIN {X -5.440, Y -12.714, Z 83.300} C_DIS
   LIN {X -5.725, Y -13.541, Z 83.300} C_DIS
   LIN {X -6.571, Y -15.942, Z 83.300} C_DIS
   LIN {X -7.033, Y -18.393, Z 83.300} C_DIS
   LIN {X -7.155, Y -19.058, Z 83.300} C_DIS
   LIN {X -7.055, Y -19.542, Z 83.300} C_DIS
   LIN {X -6.423, Y -22.696, Z 83.300} C_DIS
   LIN {X -5.056, Y -24.822, Z 83.300} C_DIS
   LIN {X -4.849, Y -25.147, Z 83.300} C_DIS
   LIN {X -4.549, Y -25.387, Z 83.300} C_DIS
   LIN {X -2.515, Y -26.991, Z 83.300} C_DIS
   LIN {X 1.598, Y -27.886, Z 83.300} C_DIS
   LIN {X 2.330, Y -28.073, Z 83.300} C_DIS
   LIN {X 2.966, Y -27.936, Z 83.300} C_DIS
   LIN {X 5.321, Y -27.375, Z 83.300} C_DIS
   LIN {X 7.789, Y -25.820, Z 83.300} C_DIS
   LIN {X 9.671, Y -23.521, Z 83.300} C_DIS
   LIN {X 10.436, Y -21.165, Z 83.300} C_DIS
   LIN {X 10.830, Y -19.986, Z 83.300} C_DIS
   LIN {X 10.937, Y -18.772, Z 83.300} C_DIS
   LIN {X 11.131, Y -16.737, Z 83.300} C_DIS
   LIN {X 11.272, Y -14.638, Z 83.300} C_DIS
   LIN {X 11.325, Y -13.783, Z 83.300} C_DIS
   LIN {X 11.361, Y -12.639, Z 83.300} C_DIS
   LIN {X 11.458, Y -9.980, Z 83.300} C_DIS
   LIN {X 11.455, Y -7.364, Z 83.300} C_DIS
   LIN {X 11.438, Y -5.193, Z 83.300} C_DIS
   LIN {X 11.377, Y -4.429, Z 83.300} C_DIS
   LIN {X 11.071, Y 1.387, Z 83.300} C_DIS
   LIN {X 9.499, Y 12.677, Z 83.300} C_DIS
   LIN {X 9.422, Y 13.171, Z 83.300} C_DIS
   LIN {X 9.298, Y 13.657, Z 83.300} C_DIS
   LIN {X 7.391, Y 21.720, Z 83.300} C_DIS
   LIN {X 6.080, Y 25.618, Z 83.300} C_DIS
   LIN {X 4.598, Y 30.349, Z 83.300} C_DIS
   LIN {X 3.927, Y 32.101, Z 83.300} C_DIS
   LIN {X 3.865, Y 32.250, Z 83.300} C_DIS
   LIN {X 3.769, Y 32.485, Z 83.300} C_DIS
   LIN {X 3.428, Y 33.345, Z 83.300} C_DIS
   LIN {X 2.495, Y 35.539, Z 83.300} C_DIS
   LIN {X 1.640, Y 37.524, Z 83.300} C_DIS
   LIN {X 0.998, Y 38.903, Z 83.300} C_DIS
   LIN {X 0.338, Y 40.306, Z 83.300} C_DIS
   LIN {X -0.759, Y 42.500, Z 83.300} C_DIS
   LIN {X -0.823, Y 42.627, Z 83.300} C_DIS
   LIN {X -0.870, Y 42.719, Z 83.300} C_DIS
   LIN {X -1.517, Y 43.955, Z 83.300} C_DIS
   LIN {X -2.348, Y 45.000, Z 83.300} C_DIS
   LIN {X -2.432, Y 45.106, Z 83.300} C_DIS
   LIN {X -2.655, Y 45.226, Z 83.300} C_DIS
   LIN {X -3.961, Y 45.935, Z 83.300} C_DIS
   LIN {X -4.774, Y 45.983, Z 83.300} C_DIS
   LIN {X -5.703, Y 46.036, Z 83.300}
   LaserEnd_Ext()
   LIN {X -3.453, Y 44.522, Z 83.300}
   LaserStart_Ext()
   LIN {X -6.351, Y 44.522, Z 83.300}
   LaserEnd_Ext()
   LIN {X -7.579, Y 43.522, Z 83.300}
   LaserStart_Ext()
   LIN {X -2.450, Y 43.522, Z 83.300}
   LaserEnd_Ext()
   LIN {X -1.896, Y 42.522, Z 83.300}
   LaserStart_Ext()
   LIN {X -7.936, Y 42.522, Z 83.300}
   LaserEnd_Ext()
   LIN {X -7.904, Y 41.522, Z 83.300}
   LaserStart_Ext()
   LIN {X -1.388, Y 41.522, Z 83.300}
   LaserEnd_Ext()
   LIN {X -0.888, Y 40.522, Z 83.300}
   LaserStart_Ext()
   LIN {X -7.596, Y 40.522, Z 83.300}
   LaserEnd_Ext()
   LIN {X -7.152, Y 39.522, Z 83.300}
   LaserStart_Ext()
   LIN {X -0.399, Y 39.522, Z 83.300}
   LaserEnd_Ext()
   LIN {X 0.072, Y 38.522, Z 83.300}
   LaserStart_Ext()
   LIN {X -6.723, Y 38.522, Z 83.300}
   LaserEnd_Ext()
   LIN {X -6.314, Y 37.522, Z 83.300}
   LaserStart_Ext()
   LIN {X 0.538, Y 37.522, Z 83.300}
   LaserEnd_Ext()
   LIN {X 0.983, Y 36.522, Z 83.300}
   LaserStart_Ext()
   LIN {X -5.917, Y 36.522, Z 83.300}
   LaserEnd_Ext()
   LIN {X -5.539, Y 35.522, Z 83.300}
   LaserStart_Ext()
   LIN {X 1.414, Y 35.522, Z 83.300}
   LaserEnd_Ext()
   LIN {X 1.841, Y 34.522, Z 83.300}
   LaserStart_Ext()
   LIN {X -5.182, Y 34.522, Z 83.300}
   LaserEnd_Ext()
   LIN {X -4.826, Y 33.522, Z 83.300}
   LaserStart_Ext()
   LIN {X 2.266, Y 33.522, Z 83.300}
   LaserEnd_Ext()
   LIN {X 2.679, Y 32.522, Z 83.300}
   LaserStart_Ext()
   LIN {X -4.500, Y 32.522, Z 83.300}
   LaserEnd_Ext()
   LIN {X -4.198, Y 31.522, Z 83.300}
   LaserStart_Ext()
   LIN {X 3.078, Y 31.522, Z 83.300}
   LaserEnd_Ext()
   LIN {X 3.461, Y 30.522, Z 83.300}
   LaserStart_Ext()
   LIN {X -3.917, Y 30.522, Z 83.300}
   LaserEnd_Ext()
   LIN {X -3.635, Y 29.522, Z 83.300}
   LaserStart_Ext()
   LIN {X 3.810, Y 29.522, Z 83.300}
   LaserEnd_Ext()
   LIN {X 4.123, Y 28.522, Z 83.300}
   LaserStart_Ext()
   LIN {X -3.354, Y 28.522, Z 83.300}
   LaserEnd_Ext()
   LIN {X -3.077, Y 27.522, Z 83.300}
   LaserStart_Ext()
   LIN {X 4.436, Y 27.522, Z 83.300}
   LaserEnd_Ext()
   LIN {X 4.749, Y 26.522, Z 83.300}
   LaserStart_Ext()
   LIN {X -2.860, Y 26.522, Z 83.300}
   LaserEnd_Ext()
   LIN {X -2.642, Y 25.522, Z 83.300}
   LaserStart_Ext()
   LIN {X 5.063, Y 25.522, Z 83.300}
   LaserEnd_Ext()
   LIN {X 5.394, Y 24.522, Z 83.300}
   LaserStart_Ext()
   LIN {X -2.425, Y 24.522, Z 83.300}
   LaserEnd_Ext()
   LIN {X -2.229, Y 23.522, Z 83.300}
   LaserStart_Ext()
   LIN {X 5.730, Y 23.522, Z 83.300}
   LaserEnd_Ext()
   LIN {X 6.067, Y 22.522, Z 83.300}
   LaserStart_Ext()
   LIN {X -2.053, Y 22.522, Z 83.300}
   LaserEnd_Ext()
   LIN {X -1.877, Y 21.522, Z 83.300}
   LaserStart_Ext()
   LIN {X 6.403, Y 21.522, Z 83.300}
   LaserEnd_Ext()
   LIN {X 6.647, Y 20.522, Z 83.300}
   LaserStart_Ext()
   LIN {X -1.724, Y 20.522, Z 83.300}
   LaserEnd_Ext()
   LIN {X -1.656, Y 19.522, Z 83.300}
   LaserStart_Ext()
   LIN {X 6.884, Y 19.522, Z 83.300}
   LaserEnd_Ext()
   LIN {X 7.120, Y 18.522, Z 83.300}
   LaserStart_Ext()
   LIN {X -1.588, Y 18.522, Z 83.300}
   LaserEnd_Ext()
   LIN {X -1.521, Y 17.522, Z 83.300}
   LaserStart_Ext()
   LIN {X 7.356, Y 17.522, Z 83.300}
   LaserEnd_Ext()
   LIN {X 7.593, Y 16.522, Z 83.300}
   LaserStart_Ext()
   LIN {X -1.453, Y 16.522, Z 83.300}
   LaserEnd_Ext()
   LIN {X -1.385, Y 15.522, Z 83.300}
   LaserStart_Ext()
   LIN {X 7.829, Y 15.522, Z 83.300}
   LaserEnd_Ext()
   LIN {X 8.066, Y 14.522, Z 83.300}
   LaserStart_Ext()
   LIN {X -1.306, Y 14.522, Z 83.300}
   LaserEnd_Ext()
   LIN {X -1.215, Y 13.522, Z 83.300}
   LaserStart_Ext()
   LIN {X 8.302, Y 13.522, Z 83.300}
   LaserEnd_Ext()
   LIN {X 8.511, Y 12.522, Z 83.300}
   LaserStart_Ext()
   LIN {X -1.124, Y 12.522, Z 83.300}
   LaserEnd_Ext()
   LIN {X -1.033, Y 11.522, Z 83.300}
   LaserStart_Ext()
   LIN {X 8.650, Y 11.522, Z 83.300}
   LaserEnd_Ext()
   LIN {X 8.790, Y 10.522, Z 83.300}
   LaserStart_Ext()
   LIN {X -0.942, Y 10.522, Z 83.300}
   LaserEnd_Ext()
   LIN {X -0.910, Y 9.522, Z 83.300}
   LaserStart_Ext()
   LIN {X 8.929, Y 9.522, Z 83.300}
   LaserEnd_Ext()
   LIN {X 9.068, Y 8.522, Z 83.300}
   LaserStart_Ext()
   LIN {X -0.908, Y 8.522, Z 83.300}
   LaserEnd_Ext()
   LIN {X -0.960, Y 7.522, Z 83.300}
   LaserStart_Ext()
   LIN {X 9.207, Y 7.522, Z 83.300}
   LaserEnd_Ext()
   LIN {X 9.347, Y 6.522, Z 83.300}
   LaserStart_Ext()
   LIN {X -1.021, Y 6.522, Z 83.300}
   LaserEnd_Ext()
   LIN {X -1.083, Y 5.522, Z 83.300}
   LaserStart_Ext()
   LIN {X 9.486, Y 5.522, Z 83.300}
   LaserEnd_Ext()
   LIN {X 9.625, Y 4.522, Z 83.300}
   LaserStart_Ext()
   LIN {X -1.145, Y 4.522, Z 83.300}
   LaserEnd_Ext()
   LIN {X -1.206, Y 3.522, Z 83.300}
   LaserStart_Ext()
   LIN {X 9.764, Y 3.522, Z 83.300}
   LaserEnd_Ext()
   LIN {X 9.903, Y 2.522, Z 83.300}
   LaserStart_Ext()
   LIN {X -1.268, Y 2.522, Z 83.300}
   LaserEnd_Ext()
   LIN {X -1.365, Y 1.522, Z 83.300}
   LaserStart_Ext()
   LIN {X 10.043, Y 1.522, Z 83.300}
   LaserEnd_Ext()
   LIN {X 10.115, Y 0.522, Z 83.300}
   LaserStart_Ext()
   LIN {X -1.462, Y 0.522, Z 83.300}
   LaserEnd_Ext()
   LIN {X -1.606, Y -0.478, Z 83.300}
   LaserStart_Ext()
   LIN {X 10.168, Y -0.478, Z 83.300}
   LaserEnd_Ext()
   LIN {X 10.220, Y -1.478, Z 83.300}
   LaserStart_Ext()
   LIN {X -1.759, Y -1.478, Z 83.300}
   LaserEnd_Ext()
   LIN {X -1.938, Y -2.478, Z 83.300}
   LaserStart_Ext()
   LIN {X 10.273, Y -2.478, Z 83.300}
   LaserEnd_Ext()
   LIN {X 10.325, Y -3.478, Z 83.300}
   LaserStart_Ext()
   LIN {X -2.116, Y -3.478, Z 83.300}
   LaserEnd_Ext()
   LIN {X -2.295, Y -4.478, Z 83.300}
   LaserStart_Ext()
   LIN {X 10.378, Y -4.478, Z 83.300}
   LaserEnd_Ext()
   LIN {X 10.440, Y -5.478, Z 83.300}
   LaserStart_Ext()
   LIN {X -2.478, Y -5.478, Z 83.300}
   LaserEnd_Ext()
   LIN {X -2.711, Y -6.478, Z 83.300}
   LaserStart_Ext()
   LIN {X 10.448, Y -6.478, Z 83.300}
   LaserEnd_Ext()
   LIN {X 10.455, Y -7.478, Z 83.300}
   LaserStart_Ext()
   LIN {X -2.955, Y -7.478, Z 83.300}
   LaserEnd_Ext()
   LIN {X -3.200, Y -8.478, Z 83.300}
   LaserStart_Ext()
   LIN {X 10.456, Y -8.478, Z 83.300}
   LaserEnd_Ext()
   LIN {X 10.457, Y -9.478, Z 83.300}
   LaserStart_Ext()
   LIN {X -3.446, Y -9.478, Z 83.300}
   LaserEnd_Ext()
   LIN {X -3.726, Y -10.478, Z 83.300}
   LaserStart_Ext()
   LIN {X 10.439, Y -10.478, Z 83.300}
   LaserEnd_Ext()
   LIN {X 10.402, Y -11.478, Z 83.300}
   LaserStart_Ext()
   LIN {X -4.027, Y -11.478, Z 83.300}
   LaserEnd_Ext()
   LIN {X -4.327, Y -12.478, Z 83.300}
   LaserStart_Ext()
   LIN {X 10.366, Y -12.478, Z 83.300}
   LaserEnd_Ext()
   LIN {X 10.334, Y -13.478, Z 83.300}
   LaserStart_Ext()
   LIN {X 3.901, Y -13.478, Z 83.300}
   LaserEnd_Ext()
   LIN {X 0.046, Y -13.478, Z 83.300}
   LaserStart_Ext()
   LIN {X -4.645, Y -13.478, Z 83.300}
   LaserEnd_Ext()
   LIN {X -4.995, Y -14.478, Z 83.300}
   LaserStart_Ext()
   LIN {X -1.898, Y -14.478, Z 83.300}
   LaserEnd_Ext()
   LIN {X 5.752, Y -14.478, Z 83.300}
   LaserStart_Ext()
   LIN {X 10.280, Y -14.478, Z 83.300}
   LaserEnd_Ext()
   LIN {X 10.214, Y -15.478, Z 83.300}
   LaserStart_Ext()
   LIN {X 6.494, Y -15.478, Z 83.300}
   LaserEnd_Ext()
   LIN {X -2.818, Y -15.478, Z 83.300}
   LaserStart_Ext()
   LIN {X -5.347, Y -15.478, Z 83.300}
   LaserEnd_Ext()
   LIN {X -5.654, Y -16.478, Z 83.300}
   LaserStart_Ext()
   LIN {X -3.444, Y -16.478, Z 83.300}
   LaserEnd_Ext()
   LIN {X 7.209, Y -16.478, Z 83.300}
   LaserStart_Ext()
   LIN {X 10.146, Y -16.478, Z 83.300}
   LaserEnd_Ext()
   LIN {X 10.056, Y -17.478, Z 83.300}
   LaserStart_Ext()
   LIN {X 7.585, Y -17.478, Z 83.300}
   LaserEnd_Ext()
   LIN {X -3.700, Y -17.478, Z 83.300}
   LaserStart_Ext()
   LIN {X -5.843, Y -17.478, Z 83.300}
   LaserEnd_Ext()
   LIN {X -6.031, Y -18.478, Z 83.300}
   LaserStart_Ext()
   LIN {X -3.953, Y -18.478, Z 83.300}
   LaserEnd_Ext()
   LIN {X 7.723, Y -18.478, Z 83.300}
   LaserStart_Ext()
   LIN {X 9.961, Y -18.478, Z 83.300}
   LaserEnd_Ext()
   LIN {X 9.871, Y -19.478, Z 83.300}
   LaserStart_Ext()
   LIN {X 7.850, Y -19.478, Z 83.300}
   LaserEnd_Ext()
   LIN {X -4.127, Y -19.478, Z 83.300}
   LaserStart_Ext()
   LIN {X -6.048, Y -19.478, Z 83.300}
   LaserEnd_Ext()
   LIN {X -5.847, Y -20.478, Z 83.300}
   LaserStart_Ext()
   LIN {X -3.874, Y -20.478, Z 83.300}
   LaserEnd_Ext()
   LIN {X 7.573, Y -20.478, Z 83.300}
   LaserStart_Ext()
   LIN {X 9.611, Y -20.478, Z 83.300}
   LaserEnd_Ext()
   LIN {X 9.283, Y -21.478, Z 83.300}
   LaserStart_Ext()
   LIN {X 7.240, Y -21.478, Z 83.300}
   LaserEnd_Ext()
   LIN {X -3.616, Y -21.478, Z 83.300}
   LaserStart_Ext()
   LIN {X -5.647, Y -21.478, Z 83.300}
   LaserEnd_Ext()
   LIN {X -5.374, Y -22.478, Z 83.300}
   LaserStart_Ext()
   LIN {X -2.994, Y -22.478, Z 83.300}
   LaserEnd_Ext()
   LIN {X 6.733, Y -22.478, Z 83.300}
   LaserStart_Ext()
   LIN {X 8.958, Y -22.478, Z 83.300}
   LaserEnd_Ext()
   LIN {X 8.417, Y -23.478, Z 83.300}
   LaserStart_Ext()
   LIN {X 5.780, Y -23.478, Z 83.300}
   LaserEnd_Ext()
   LIN {X -2.183, Y -23.478, Z 83.300}
   LaserStart_Ext()
   LIN {X -4.731, Y -23.478, Z 83.300}
   LaserEnd_Ext()
   LIN {X -4.085, Y -24.478, Z 83.300}
   LaserStart_Ext()
   LIN {X -0.558, Y -24.478, Z 83.300}
   LaserEnd_Ext()
   LIN {X 4.172, Y -24.478, Z 83.300}
   LaserStart_Ext()
   LIN {X 7.605, Y -24.478, Z 83.300}
   LaserEnd_Ext()
   LIN {X 6.455, Y -25.478, Z 83.300}
   LaserStart_Ext()
   LIN {X -2.818, Y -25.478, Z 83.300}
   LaserEnd_Ext()
   LIN {X -0.167, Y -26.478, Z 83.300}
   LaserStart_Ext()
   LIN {X 4.769, Y -26.478, Z 83.300}
   LaserEnd_Ext()
   LIN {X -2.559, Y -21.198, Z 84.150}
   LaserStart_Ext()
   LIN {X -3.058, Y -19.292, Z 84.150} C_DIS
   LIN {X -2.579, Y -17.398, Z 84.150} C_DIS
   LIN {X -2.354, Y -16.480, Z 84.150} C_DIS
   LIN {X -1.630, Y -15.678, Z 84.150} C_DIS
   LIN {X -0.982, Y -14.973, Z 84.150} C_DIS
   LIN {X -0.310, Y -14.697, Z 84.150} C_DIS
   LIN {X 1.140, Y -14.083, Z 84.150} C_DIS
   LIN {X 3.021, Y -14.162, Z 84.150} C_DIS
   LIN {X 3.247, Y -14.172, Z 84.150} C_DIS
   LIN {X 3.412, Y -14.257, Z 84.150} C_DIS
   LIN {X 5.138, Y -15.143, Z 84.150} C_DIS
   LIN {X 6.591, Y -17.162, Z 84.150} C_DIS
   LIN {X 6.631, Y -17.256, Z 84.150} C_DIS
   LIN {X 6.932, Y -19.395, Z 84.150} C_DIS
   LIN {X 6.243, Y -21.534, Z 84.150} C_DIS
   LIN {X 4.736, Y -23.156, Z 84.150} C_DIS
   LIN {X 3.536, Y -23.634, Z 84.150} C_DIS
   LIN {X 2.696, Y -23.962, Z 84.150} C_DIS
   LIN {X 1.432, Y -23.900, Z 84.150} C_DIS
   LIN {X 0.627, Y -23.863, Z 84.150} C_DIS
   LIN {X 0.122, Y -23.608, Z 84.150} C_DIS
   LIN {X -1.215, Y -22.926, Z 84.150} C_DIS
   LIN {X -2.449, Y -21.408, Z 84.150} C_DIS
   LIN {X -2.529, Y -21.310, Z 84.150} C_DIS
   LIN {X -2.559, Y -21.198, Z 84.150}
   LaserEnd_Ext()
   LIN {X -1.905, Y 7.936, Z 84.150}
   LaserStart_Ext()
   LIN {X -2.220, Y 2.830, Z 84.150} C_DIS
   LIN {X -2.462, Y 0.323, Z 84.150} C_DIS
   LIN {X -2.793, Y -1.838, Z 84.150} C_DIS
   LIN {X -3.215, Y -4.200, Z 84.150} C_DIS
   LIN {X -3.484, Y -5.603, Z 84.150} C_DIS
   LIN {X -4.244, Y -8.736, Z 84.150} C_DIS
   LIN {X -4.440, Y -9.531, Z 84.150} C_DIS
   LIN {X -4.630, Y -10.161, Z 84.150} C_DIS
   LIN {X -5.341, Y -12.571, Z 84.150} C_DIS
   LIN {X -6.198, Y -15.055, Z 84.150} C_DIS
   LIN {X -6.498, Y -15.906, Z 84.150} C_DIS
   LIN {X -6.662, Y -16.775, Z 84.150} C_DIS
   LIN {X -7.075, Y -19.024, Z 84.150} C_DIS
   LIN {X -6.736, Y -20.655, Z 84.150} C_DIS
   LIN {X -6.334, Y -22.659, Z 84.150} C_DIS
   LIN {X -5.189, Y -24.441, Z 84.150} C_DIS
   LIN {X -4.755, Y -25.107, Z 84.150} C_DIS
   LIN {X -3.600, Y -26.012, Z 84.150} C_DIS
   LIN {X -2.416, Y -26.945, Z 84.150} C_DIS
   LIN {X 0.336, Y -27.544, Z 84.150} C_DIS
   LIN {X 2.444, Y -28.017, Z 84.150} C_DIS
   LIN {X 3.075, Y -27.886, Z 84.150} C_DIS
   LIN {X 5.333, Y -27.347, Z 84.150} C_DIS
   LIN {X 6.980, Y -26.310, Z 84.150} C_DIS
   LIN {X 7.837, Y -25.797, Z 84.150} C_DIS
   LIN {X 8.738, Y -24.731, Z 84.150} C_DIS
   LIN {X 9.716, Y -23.527, Z 84.150} C_DIS
   LIN {X 10.125, Y -22.267, Z 84.150} C_DIS
   LIN {X 10.912, Y -19.908, Z 84.150} C_DIS
   LIN {X 11.128, Y -17.481, Z 84.150} C_DIS
   LIN {X 11.206, Y -16.659, Z 84.150} C_DIS
   LIN {X 11.263, Y -15.811, Z 84.150} C_DIS
   LIN {X 11.393, Y -13.704, Z 84.150} C_DIS
   LIN {X 11.481, Y -10.887, Z 84.150} C_DIS
   LIN {X 11.517, Y -9.901, Z 84.150} C_DIS
   LIN {X 11.516, Y -8.932, Z 84.150} C_DIS
   LIN {X 11.486, Y -5.114, Z 84.150} C_DIS
   LIN {X 11.378, Y -3.771, Z 84.150} C_DIS
   LIN {X 11.102, Y 1.481, Z 84.150} C_DIS
   LIN {X 9.682, Y 11.678, Z 84.150} C_DIS
   LIN {X 9.461, Y 13.085, Z 84.150} C_DIS
   LIN {X 9.108, Y 14.470, Z 84.150} C_DIS
   LIN {X 7.387, Y 21.750, Z 84.150} C_DIS
   LIN {X 5.820, Y 26.408, Z 84.150} C_DIS
   LIN {X 4.596, Y 30.316, Z 84.150} C_DIS
   LIN {X 4.042, Y 31.764, Z 84.150} C_DIS
   LIN {X 3.990, Y 31.887, Z 84.150} C_DIS
   LIN {X 3.911, Y 32.081, Z 84.150} C_DIS
   LIN {X 3.466, Y 33.203, Z 84.150} C_DIS
   LIN {X 2.958, Y 34.398, Z 84.150} C_DIS
   LIN {X 1.589, Y 37.576, Z 84.150} C_DIS
   LIN {X 1.428, Y 37.916, Z 84.150} C_DIS
   LIN {X 0.343, Y 40.225, Z 84.150} C_DIS
   LIN {X 0.034, Y 40.842, Z 84.150} C_DIS
   LIN {X -0.891, Y 42.682, Z 84.150} C_DIS
   LIN {X -1.581, Y 43.994, Z 84.150} C_DIS
   LIN {X -2.503, Y 45.151, Z 84.150} C_DIS
   LIN {X -3.508, Y 45.694, Z 84.150} C_DIS
   LIN {X -4.034, Y 45.976, Z 84.150} C_DIS
   LIN {X -4.951, Y 46.027, Z 84.150} C_DIS
   LIN {X -5.776, Y 46.074, Z 84.150} C_DIS
   LIN {X -6.543, Y 45.640, Z 84.150} C_DIS
   LIN {X -8.156, Y 44.716, Z 84.150} C_DIS
   LIN {X -8.853, Y 43.436, Z 84.150} C_DIS
   LIN {X -8.922, Y 43.309, Z 84.150} C_DIS
   LIN {X -8.935, Y 43.190, Z 84.150} C_DIS
   LIN {X -9.082, Y 41.866, Z 84.150} C_DIS
   LIN {X -8.799, Y 40.795, Z 84.150} C_DIS
   LIN {X -8.711, Y 40.461, Z 84.150} C_DIS
   LIN {X -8.530, Y 40.058, Z 84.150} C_DIS
   LIN {X -8.198, Y 39.321, Z 84.150} C_DIS
   LIN {X -7.964, Y 38.782, Z 84.150} C_DIS
   LIN {X -7.563, Y 37.853, Z 84.150} C_DIS
   LIN {X -6.793, Y 35.927, Z 84.150} C_DIS
   LIN {X -6.683, Y 35.652, Z 84.150} C_DIS
   LIN {X -6.569, Y 35.338, Z 84.150} C_DIS
   LIN {X -5.711, Y 32.948, Z 84.150} C_DIS
   LIN {X -5.428, Y 32.041, Z 84.150} C_DIS
   LIN {X -5.095, Y 30.976, Z 84.150} C_DIS
   LIN {X -4.152, Y 27.623, Z 84.150} C_DIS
   LIN {X -3.127, Y 22.913, Z 84.150} C_DIS
   LIN {X -2.784, Y 20.964, Z 84.150} C_DIS
   LIN {X -2.553, Y 17.560, Z 84.150} C_DIS
   LIN {X -1.910, Y 10.485, Z 84.150} C_DIS
   LIN {X -1.905, Y 7.936, Z 84.150}
   LaserEnd_Ext()
   LIN {X -7.280, Y 39.718, Z 84.150}
   LaserStart_Ext()
   LIN {X -7.280, Y 44.065, Z 84.150}
   LaserEnd_Ext()
   LIN {X -6.280, Y 44.639, Z 84.150}
   LaserStart_Ext()
   LIN {X -6.280, Y 37.336, Z 84.150}
   LaserEnd_Ext()
   LIN {X -5.280, Y -22.450, Z 84.150}
   LaserStart_Ext()
   LIN {X -5.280, Y -15.458, Z 84.150}
   LaserEnd_Ext()
   LIN {X -5.280, Y 34.706, Z 84.150}
   LaserStart_Ext()
   LIN {X -5.280, Y 45.044, Z 84.150}
   LaserEnd_Ext()
   LIN {X -4.280, Y 44.973, Z 84.150}
   LaserStart_Ext()
   LIN {X -4.280, Y 31.720, Z 84.150}
   LaserEnd_Ext()
   LIN {X -4.280, Y -12.507, Z 84.150}
   LaserStart_Ext()
   LIN {X -4.280, Y -24.005, Z 84.150}
   LaserEnd_Ext()
   LIN {X -3.280, Y -24.993, Z 84.150}
   LaserStart_Ext()
   LIN {X -3.280, Y -21.972, Z 84.150}
   LaserEnd_Ext()
   LIN {X -3.280, Y -16.106, Z 84.150}
   LaserStart_Ext()
   LIN {X -3.280, Y -9.001, Z 84.150}
   LaserEnd_Ext()
   LIN {X -3.280, Y 28.216, Z 84.150}
   LaserStart_Ext()
   LIN {X -3.280, Y 44.434, Z 84.150}
   LaserEnd_Ext()
   LIN {X -2.280, Y 43.175, Z 84.150}
   LaserStart_Ext()
   LIN {X -2.280, Y 23.722, Z 84.150}
   LaserEnd_Ext()
   LIN {X -2.280, Y -4.635, Z 84.150}
   LaserStart_Ext()
   LIN {X -2.280, Y -14.907, Z 84.150}
   LaserEnd_Ext()
   LIN {X -2.280, Y -23.201, Z 84.150}
   LaserStart_Ext()
   LIN {X -2.280, Y -25.779, Z 84.150}
   LaserEnd_Ext()
   LIN {X -1.280, Y -26.169, Z 84.150}
   LaserStart_Ext()
   LIN {X -1.280, Y -24.015, Z 84.150}
   LaserEnd_Ext()
   LIN {X -1.280, Y -14.014, Z 84.150}
   LaserStart_Ext()
   LIN {X -1.280, Y 2.162, Z 84.150}
   LaserEnd_Ext()
   LIN {X -1.280, Y 14.596, Z 84.150}
   LaserStart_Ext()
   LIN {X -1.280, Y 41.230, Z 84.150}
   LaserEnd_Ext()
   LIN {X -0.280, Y 39.199, Z 84.150}
   LaserStart_Ext()
   LIN {X -0.280, Y -13.598, Z 84.150}
   LaserEnd_Ext()
   LIN {X -0.280, Y -24.525, Z 84.150}
   LaserStart_Ext()
   LIN {X -0.280, Y -26.387, Z 84.150}
   LaserEnd_Ext()
   LIN {X 0.720, Y -26.606, Z 84.150}
   LaserStart_Ext()
   LIN {X 0.720, Y -24.868, Z 84.150}
   LaserEnd_Ext()
   LIN {X 0.720, Y -13.175, Z 84.150}
   LaserStart_Ext()
   LIN {X 0.720, Y 37.064, Z 84.150}
   LaserEnd_Ext()
   LIN {X 1.720, Y 34.743, Z 84.150}
   LaserStart_Ext()
   LIN {X 1.720, Y -13.107, Z 84.150}
   LaserEnd_Ext()
   LIN {X 1.720, Y -24.915, Z 84.150}
   LaserStart_Ext()
   LIN {X 1.720, Y -26.830, Z 84.150}
   LaserEnd_Ext()
   LIN {X 2.720, Y -26.939, Z 84.150}
   LaserStart_Ext()
   LIN {X 2.720, Y -24.960, Z 84.150}
   LaserEnd_Ext()
   LIN {X 2.720, Y -13.148, Z 84.150}
   LaserStart_Ext()
   LIN {X 2.720, Y 32.371, Z 84.150}
   LaserEnd_Ext()
   LIN {X 3.720, Y 29.767, Z 84.150}
   LaserStart_Ext()
   LIN {X 3.720, Y -13.290, Z 84.150}
   LaserEnd_Ext()
   LIN {X 3.720, Y -24.635, Z 84.150}
   LaserStart_Ext()
   LIN {X 3.720, Y -26.704, Z 84.150}
   LaserEnd_Ext()
   LIN {X 4.720, Y -26.466, Z 84.150}
   LaserStart_Ext()
   LIN {X 4.720, Y -24.239, Z 84.150}
   LaserEnd_Ext()
   LIN {X 4.720, Y -13.804, Z 84.150}
   LaserStart_Ext()
   LIN {X 4.720, Y 26.575, Z 84.150}
   LaserEnd_Ext()
   LIN {X 5.720, Y 23.569, Z 84.150}
   LaserStart_Ext()
   LIN {X 5.720, Y -14.331, Z 84.150}
   LaserEnd_Ext()
   LIN {X 5.720, Y -23.570, Z 84.150}
   LaserStart_Ext()
   LIN {X 5.720, Y -25.922, Z 84.150}
   LaserEnd_Ext()
   LIN {X 6.720, Y -25.300, Z 84.150}
   LaserStart_Ext()
   LIN {X 6.720, Y -22.506, Z 84.150}
   LaserEnd_Ext()
   LIN {X 6.720, Y -15.630, Z 84.150}
   LaserStart_Ext()
   LIN {X 6.720, Y 20.224, Z 84.150}
   LaserEnd_Ext()
   LIN {X 7.720, Y 15.994, Z 84.150}
   LaserStart_Ext()
   LIN {X 7.720, Y -17.822, Z 84.150}
   LaserEnd_Ext()
   LIN {X 7.720, Y -20.210, Z 84.150}
   LaserStart_Ext()
   LIN {X 7.720, Y -24.386, Z 84.150}
   LaserEnd_Ext()
   LIN {X 8.720, Y -23.167, Z 84.150}
   LaserStart_Ext()
   LIN {X 8.720, Y 11.335, Z 84.150}
   LaserEnd_Ext()
   LIN {X 9.720, Y 4.152, Z 84.150}
   LaserStart_Ext()
   LIN {X 9.720, Y -20.321, Z 84.150}
   LaserEnd_Ext()
   LIN {X -2.285, Y -16.444, Z 85.000}
   LaserStart_Ext()
   LIN {X -1.288, Y -15.338, Z 85.000} C_DIS
   LIN {X -0.949, Y -14.951, Z 85.000} C_DIS
   LIN {X -0.125, Y -14.596, Z 85.000} C_DIS
   LIN {X 1.216, Y -14.028, Z 85.000} C_DIS
   LIN {X 2.191, Y -14.068, Z 85.000} C_DIS
   LIN {X 3.316, Y -14.112, Z 85.000} C_DIS
   LIN {X 4.625, Y -14.780, Z 85.000} C_DIS
   LIN {X 5.209, Y -15.079, Z 85.000} C_DIS
   LIN {X 5.612, Y -15.640, Z 85.000} C_DIS
   LIN {X 6.699, Y -17.139, Z 85.000} C_DIS
   LIN {X 6.939, Y -18.803, Z 85.000} C_DIS
   LIN {X 7.013, Y -19.327, Z 85.000} C_DIS
   LIN {X 6.840, Y -19.866, Z 85.000} C_DIS
   LIN {X 6.321, Y -21.496, Z 85.000} C_DIS
   LIN {X 5.500, Y -22.377, Z 85.000} C_DIS
   LIN {X 4.828, Y -23.092, Z 85.000} C_DIS
   LIN {X 3.329, Y -23.689, Z 85.000} C_DIS
   LIN {X 2.796, Y -23.902, Z 85.000} C_DIS
   LIN {X 2.441, Y -23.888, Z 85.000} C_DIS
   LIN {X 0.719, Y -23.810, Z 85.000} C_DIS
   LIN {X -0.902, Y -22.991, Z 85.000} C_DIS
   LIN {X -1.125, Y -22.877, Z 85.000} C_DIS
   LIN {X -1.332, Y -22.624, Z 85.000} C_DIS
   LIN {X -2.444, Y -21.265, Z 85.000} C_DIS
   LIN {X -2.859, Y -19.699, Z 85.000} C_DIS
   LIN {X -2.977, Y -19.248, Z 85.000} C_DIS
   LIN {X -2.863, Y -18.799, Z 85.000} C_DIS
   LIN {X -2.285, Y -16.444, Z 85.000}
   LaserEnd_Ext()
   LIN {X 0.677, Y 39.452, Z 85.000}
   LaserStart_Ext()
   LIN {X 1.537, Y 37.627, Z 85.000} C_DIS
   LIN {X 3.420, Y 33.257, Z 85.000} C_DIS
   LIN {X 3.504, Y 33.061, Z 85.000} C_DIS
   LIN {X 4.053, Y 31.677, Z 85.000} C_DIS
   LIN {X 4.115, Y 31.524, Z 85.000} C_DIS
   LIN {X 4.156, Y 31.427, Z 85.000} C_DIS
   LIN {X 4.594, Y 30.284, Z 85.000} C_DIS
   LIN {X 5.560, Y 27.197, Z 85.000} C_DIS
   LIN {X 7.382, Y 21.780, Z 85.000} C_DIS
   LIN {X 8.919, Y 15.282, Z 85.000} C_DIS
   LIN {X 9.501, Y 12.998, Z 85.000} C_DIS
   LIN {X 9.865, Y 10.679, Z 85.000} C_DIS
   LIN {X 11.132, Y 1.576, Z 85.000} C_DIS
   LIN {X 11.379, Y -3.113, Z 85.000} C_DIS
   LIN {X 11.534, Y -5.036, Z 85.000} C_DIS
   LIN {X 11.558, Y -8.170, Z 85.000} C_DIS
   LIN {X 11.576, Y -9.823, Z 85.000} C_DIS
   LIN {X 11.563, Y -10.352, Z 85.000} C_DIS
   LIN {X 11.461, Y -13.626, Z 85.000} C_DIS
   LIN {X 11.299, Y -16.248, Z 85.000} C_DIS
   LIN {X 11.281, Y -16.581, Z 85.000} C_DIS
   LIN {X 11.249, Y -16.971, Z 85.000} C_DIS
   LIN {X 10.995, Y -19.831, Z 85.000} C_DIS
   LIN {X 9.814, Y -23.369, Z 85.000} C_DIS
   LIN {X 9.760, Y -23.533, Z 85.000} C_DIS
   LIN {X 9.633, Y -23.690, Z 85.000} C_DIS
   LIN {X 7.859, Y -25.790, Z 85.000} C_DIS
   LIN {X 6.170, Y -26.800, Z 85.000} C_DIS
   LIN {X 5.345, Y -27.320, Z 85.000} C_DIS
   LIN {X 4.214, Y -27.590, Z 85.000} C_DIS
   LIN {X 2.401, Y -27.966, Z 85.000} C_DIS
   LIN {X -1.841, Y -27.015, Z 85.000} C_DIS
   LIN {X -2.317, Y -26.899, Z 85.000} C_DIS
   LIN {X -2.605, Y -26.677, Z 85.000} C_DIS
   LIN {X -4.660, Y -25.067, Z 85.000} C_DIS
   LIN {X -5.758, Y -23.382, Z 85.000} C_DIS
   LIN {X -6.246, Y -22.623, Z 85.000} C_DIS
   LIN {X -6.417, Y -21.768, Z 85.000} C_DIS
   LIN {X -6.994, Y -18.989, Z 85.000} C_DIS
   LIN {X -6.507, Y -16.333, Z 85.000} C_DIS
   LIN {X -6.425, Y -15.870, Z 85.000} C_DIS
   LIN {X -6.173, Y -15.124, Z 85.000} C_DIS
   LIN {X -5.243, Y -12.427, Z 85.000} C_DIS
   LIN {X -4.588, Y -10.211, Z 85.000} C_DIS
   LIN {X -4.374, Y -9.461, Z 85.000} C_DIS
   LIN {X -4.204, Y -8.748, Z 85.000} C_DIS
   LIN {X -3.472, Y -5.734, Z 85.000} C_DIS
   LIN {X -3.037, Y -3.468, Z 85.000} C_DIS
   LIN {X -2.839, Y -2.358, Z 85.000} C_DIS
   LIN {X -2.456, Y 0.149, Z 85.000} C_DIS
   LIN {X -2.175, Y 3.057, Z 85.000} C_DIS
   LIN {X -1.902, Y 7.474, Z 85.000} C_DIS
   LIN {X -1.909, Y 10.835, Z 85.000} C_DIS
   LIN {X -2.757, Y 20.161, Z 85.000} C_DIS
   LIN {X -2.835, Y 21.311, Z 85.000} C_DIS
   LIN {X -2.951, Y 21.970, Z 85.000} C_DIS
   LIN {X -4.239, Y 27.892, Z 85.000} C_DIS
   LIN {X -4.938, Y 30.376, Z 85.000} C_DIS
   LIN {X -5.184, Y 31.165, Z 85.000} C_DIS
   LIN {X -5.708, Y 32.838, Z 85.000} C_DIS
   LIN {X -5.766, Y 33.023, Z 85.000} C_DIS
   LIN {X -5.939, Y 33.498, Z 85.000} C_DIS
   LIN {X -6.731, Y 35.687, Z 85.000} C_DIS
   LIN {X -7.398, Y 37.346, Z 85.000} C_DIS
   LIN {X -7.617, Y 37.886, Z 85.000} C_DIS
   LIN {X -7.763, Y 38.220, Z 85.000} C_DIS
   LIN {X -8.255, Y 39.353, Z 85.000} C_DIS
   LIN {X -8.487, Y 39.867, Z 85.000} C_DIS
   LIN {X -8.771, Y 40.492, Z 85.000} C_DIS
   LIN {X -9.073, Y 41.633, Z 85.000} C_DIS
   LIN {X -9.146, Y 41.906, Z 85.000} C_DIS
   LIN {X -9.120, Y 42.139, Z 85.000} C_DIS
   LIN {X -9.002, Y 43.293, Z 85.000} C_DIS
   LIN {X -8.425, Y 44.391, Z 85.000} C_DIS
   LIN {X -8.242, Y 44.727, Z 85.000} C_DIS
   LIN {X -7.491, Y 45.158, Z 85.000} C_DIS
   LIN {X -5.849, Y 46.111, Z 85.000} C_DIS
   LIN {X -4.979, Y 46.066, Z 85.000} C_DIS
   LIN {X -4.107, Y 46.018, Z 85.000} C_DIS
   LIN {X -2.966, Y 45.406, Z 85.000} C_DIS
   LIN {X -2.574, Y 45.196, Z 85.000} C_DIS
   LIN {X -2.391, Y 44.969, Z 85.000} C_DIS
   LIN {X -1.653, Y 44.050, Z 85.000} C_DIS
   LIN {X -1.007, Y 42.829, Z 85.000} C_DIS
   LIN {X -0.952, Y 42.724, Z 85.000} C_DIS
   LIN {X -0.808, Y 42.437, Z 85.000} C_DIS
   LIN {X 0.237, Y 40.368, Z 85.000} C_DIS
   LIN {X 0.677, Y 39.452, Z 85.000}
   LaserEnd_Ext()
   LIN {X 4.993, Y -26.360, Z 85.000}
   LaserStart_Ext()
   LIN {X -0.191, Y -26.360, Z 85.000}
   LaserEnd_Ext()
   LIN {X -2.664, Y -25.360, Z 85.000}
   LaserStart_Ext()
   LIN {X 6.630, Y -25.360, Z 85.000}
   LaserEnd_Ext()
   LIN {X 7.758, Y -24.360, Z 85.000}
   LaserStart_Ext()
   LIN {X 4.346, Y -24.360, Z 85.000}
   LaserEnd_Ext()
   LIN {X -0.410, Y -24.360, Z 85.000}
   LaserStart_Ext()
   LIN {X -3.927, Y -24.360, Z 85.000}
   LaserEnd_Ext()
   LIN {X -4.579, Y -23.360, Z 85.000}
   LaserStart_Ext()
   LIN {X -2.022, Y -23.360, Z 85.000}
   LaserEnd_Ext()
   LIN {X 5.949, Y -23.360, Z 85.000}
   LaserStart_Ext()
   LIN {X 8.603, Y -23.360, Z 85.000}
   LaserEnd_Ext()
   LIN {X 9.096, Y -22.360, Z 85.000}
   LaserStart_Ext()
   LIN {X 6.883, Y -22.360, Z 85.000}
   LaserEnd_Ext()
   LIN {X -2.840, Y -22.360, Z 85.000}
   LaserStart_Ext()
   LIN {X -5.226, Y -22.360, Z 85.000}
   LaserEnd_Ext()
   LIN {X -5.480, Y -21.360, Z 85.000}
   LaserStart_Ext()
   LIN {X -3.453, Y -21.360, Z 85.000}
   LaserEnd_Ext()
   LIN {X 7.413, Y -21.360, Z 85.000}
   LaserStart_Ext()
   LIN {X 9.430, Y -21.360, Z 85.000}
   LaserEnd_Ext()
   LIN {X 9.764, Y -20.360, Z 85.000}
   LaserStart_Ext()
   LIN {X 7.732, Y -20.360, Z 85.000}
   LaserEnd_Ext()
   LIN {X -3.718, Y -20.360, Z 85.000}
   LaserStart_Ext()
   LIN {X -5.688, Y -20.360, Z 85.000}
   LaserEnd_Ext()
   LIN {X -5.896, Y -19.360, Z 85.000}
   LaserStart_Ext()
   LIN {X -3.969, Y -19.360, Z 85.000}
   LaserEnd_Ext()
   LIN {X 8.012, Y -19.360, Z 85.000}
   LaserStart_Ext()
   LIN {X 10.033, Y -19.360, Z 85.000}
   LaserEnd_Ext()
   LIN {X 10.122, Y -18.360, Z 85.000}
   LaserStart_Ext()
   LIN {X 7.886, Y -18.360, Z 85.000}
   LaserEnd_Ext()
   LIN {X -3.786, Y -18.360, Z 85.000}
   LaserStart_Ext()
   LIN {X -5.862, Y -18.360, Z 85.000}
   LaserEnd_Ext()
   LIN {X -5.679, Y -17.360, Z 85.000}
   LaserStart_Ext()
   LIN {X -3.540, Y -17.360, Z 85.000}
   LaserEnd_Ext()
   LIN {X 7.742, Y -17.360, Z 85.000}
   LaserStart_Ext()
   LIN {X 10.210, Y -17.360, Z 85.000}
   LaserEnd_Ext()
   LIN {X 10.292, Y -16.360, Z 85.000}
   LaserStart_Ext()
   LIN {X 7.370, Y -16.360, Z 85.000}
   LaserEnd_Ext()
   LIN {X -3.295, Y -16.360, Z 85.000}
   LaserStart_Ext()
   LIN {X -5.496, Y -16.360, Z 85.000}
   LaserEnd_Ext()
   LIN {X -5.197, Y -15.360, Z 85.000}
   LaserStart_Ext()
   LIN {X -2.655, Y -15.360, Z 85.000}
   LaserEnd_Ext()
   LIN {X 6.645, Y -15.360, Z 85.000}
   LaserStart_Ext()
   LIN {X 10.352, Y -15.360, Z 85.000}
   LaserEnd_Ext()
   LIN {X 10.414, Y -14.360, Z 85.000}
   LaserStart_Ext()
   LIN {X 5.903, Y -14.360, Z 85.000}
   LaserEnd_Ext()
   LIN {X -1.760, Y -14.360, Z 85.000}
   LaserStart_Ext()
   LIN {X -4.852, Y -14.360, Z 85.000}
   LaserEnd_Ext()
   LIN {X -4.507, Y -13.360, Z 85.000}
   LaserStart_Ext()
   LIN {X 0.228, Y -13.360, Z 85.000}
   LaserEnd_Ext()
   LIN {X 4.042, Y -13.360, Z 85.000}
   LaserStart_Ext()
   LIN {X 10.469, Y -13.360, Z 85.000}
   LaserEnd_Ext()
   LIN {X 10.500, Y -12.360, Z 85.000}
   LaserStart_Ext()
   LIN {X -4.181, Y -12.360, Z 85.000}
   LaserEnd_Ext()
   LIN {X -3.885, Y -11.360, Z 85.000}
   LaserStart_Ext()
   LIN {X 10.531, Y -11.360, Z 85.000}
   LaserEnd_Ext()
   LIN {X 10.562, Y -10.360, Z 85.000}
   LaserStart_Ext()
   LIN {X -3.591, Y -10.360, Z 85.000}
   LaserEnd_Ext()
   LIN {X -3.322, Y -9.360, Z 85.000}
   LaserStart_Ext()
   LIN {X 10.571, Y -9.360, Z 85.000}
   LaserEnd_Ext()
   LIN {X 10.560, Y -8.360, Z 85.000}
   LaserStart_Ext()
   LIN {X -3.080, Y -8.360, Z 85.000}
   LaserEnd_Ext()
   LIN {X -2.837, Y -7.360, Z 85.000}
   LaserStart_Ext()
   LIN {X 10.552, Y -7.360, Z 85.000}
   LaserEnd_Ext()
   LIN {X 10.544, Y -6.360, Z 85.000}
   LaserStart_Ext()
   LIN {X -2.595, Y -6.360, Z 85.000}
   LaserEnd_Ext()
   LIN {X -2.382, Y -5.360, Z 85.000}
   LaserStart_Ext()
   LIN {X 10.536, Y -5.360, Z 85.000}
   LaserEnd_Ext()
   LIN {X 10.476, Y -4.360, Z 85.000}
   LaserStart_Ext()
   LIN {X -2.190, Y -4.360, Z 85.000}
   LaserEnd_Ext()
   LIN {X -2.002, Y -3.360, Z 85.000}
   LaserStart_Ext()
   LIN {X 10.395, Y -3.360, Z 85.000}
   LaserEnd_Ext()
   LIN {X 10.338, Y -2.360, Z 85.000}
   LaserStart_Ext()
   LIN {X -1.828, Y -2.360, Z 85.000}
   LaserEnd_Ext()
   LIN {X -1.675, Y -1.360, Z 85.000}
   LaserStart_Ext()
   LIN {X 10.285, Y -1.360, Z 85.000}
   LaserEnd_Ext()
   LIN {X 10.233, Y -0.360, Z 85.000}
   LaserStart_Ext()
   LIN {X -1.522, Y -0.360, Z 85.000}
   LaserEnd_Ext()
   LIN {X -1.404, Y 0.640, Z 85.000}
   LaserStart_Ext()
   LIN {X 10.180, Y 0.640, Z 85.000}
   LaserEnd_Ext()
   LIN {X 10.114, Y 1.640, Z 85.000}
   LaserStart_Ext()
   LIN {X -1.307, Y 1.640, Z 85.000}
   LaserEnd_Ext()
   LIN {X -1.210, Y 2.640, Z 85.000}
   LaserStart_Ext()
   LIN {X 9.974, Y 2.640, Z 85.000}
   LaserEnd_Ext()
   LIN {X 9.835, Y 3.640, Z 85.000}
   LaserStart_Ext()
   LIN {X -1.137, Y 3.640, Z 85.000}
   LaserEnd_Ext()
   LIN {X -1.075, Y 4.640, Z 85.000}
   LaserStart_Ext()
   LIN {X 9.696, Y 4.640, Z 85.000}
   LaserEnd_Ext()
   LIN {X 9.557, Y 5.640, Z 85.000}
   LaserStart_Ext()
   LIN {X -1.013, Y 5.640, Z 85.000}
   LaserEnd_Ext()
   LIN {X -0.952, Y 6.640, Z 85.000}
   LaserStart_Ext()
   LIN {X 9.418, Y 6.640, Z 85.000}
   LaserEnd_Ext()
   LIN {X 9.278, Y 7.640, Z 85.000}
   LaserStart_Ext()
   LIN {X -0.903, Y 7.640, Z 85.000}
   LaserEnd_Ext()
   LIN {X -0.905, Y 8.640, Z 85.000}
   LaserStart_Ext()
   LIN {X 9.139, Y 8.640, Z 85.000}
   LaserEnd_Ext()
   LIN {X 9.000, Y 9.640, Z 85.000}
   LaserStart_Ext()
   LIN {X -0.907, Y 9.640, Z 85.000}
   LaserEnd_Ext()
   LIN {X -0.909, Y 10.640, Z 85.000}
   LaserStart_Ext()
   LIN {X 8.859, Y 10.640, Z 85.000}
   LaserEnd_Ext()
   LIN {X 8.702, Y 11.640, Z 85.000}
   LaserStart_Ext()
   LIN {X -0.978, Y 11.640, Z 85.000}
   LaserEnd_Ext()
   LIN {X -1.069, Y 12.640, Z 85.000}
   LaserStart_Ext()
   LIN {X 8.545, Y 12.640, Z 85.000}
   LaserEnd_Ext()
   LIN {X 8.305, Y 13.640, Z 85.000}
   LaserStart_Ext()
   LIN {X -1.160, Y 13.640, Z 85.000}
   LaserEnd_Ext()
   LIN {X -1.251, Y 14.640, Z 85.000}
   LaserStart_Ext()
   LIN {X 8.050, Y 14.640, Z 85.000}
   LaserEnd_Ext()
   LIN {X 7.807, Y 15.640, Z 85.000}
   LaserStart_Ext()
   LIN {X -1.342, Y 15.640, Z 85.000}
   LaserEnd_Ext()
   LIN {X -1.433, Y 16.640, Z 85.000}
   LaserStart_Ext()
   LIN {X 7.570, Y 16.640, Z 85.000}
   LaserEnd_Ext()
   LIN {X 7.334, Y 17.640, Z 85.000}
   LaserStart_Ext()
   LIN {X -1.524, Y 17.640, Z 85.000}
   LaserEnd_Ext()
   LIN {X -1.615, Y 18.640, Z 85.000}
   LaserStart_Ext()
   LIN {X 7.097, Y 18.640, Z 85.000}
   LaserEnd_Ext()
   LIN {X 6.861, Y 19.640, Z 85.000}
   LaserStart_Ext()
   LIN {X -1.706, Y 19.640, Z 85.000}
   LaserEnd_Ext()
   LIN {X -1.787, Y 20.640, Z 85.000}
   LaserStart_Ext()
   LIN {X 6.624, Y 20.640, Z 85.000}
   LaserEnd_Ext()
   LIN {X 6.374, Y 21.640, Z 85.000}
   LaserStart_Ext()
   LIN {X -1.878, Y 21.640, Z 85.000}
   LaserEnd_Ext()
   LIN {X -2.074, Y 22.640, Z 85.000}
   LaserStart_Ext()
   LIN {X 6.038, Y 22.640, Z 85.000}
   LaserEnd_Ext()
   LIN {X 5.702, Y 23.640, Z 85.000}
   LaserStart_Ext()
   LIN {X -2.291, Y 23.640, Z 85.000}
   LaserEnd_Ext()
   LIN {X -2.509, Y 24.640, Z 85.000}
   LaserStart_Ext()
   LIN {X 5.366, Y 24.640, Z 85.000}
   LaserEnd_Ext()
   LIN {X 5.029, Y 25.640, Z 85.000}
   LaserStart_Ext()
   LIN {X -2.726, Y 25.640, Z 85.000}
   LaserEnd_Ext()
   LIN {X -2.944, Y 26.640, Z 85.000}
   LaserStart_Ext()
   LIN {X 4.693, Y 26.640, Z 85.000}
   LaserEnd_Ext()
   LIN {X 4.374, Y 27.640, Z 85.000}
   LaserStart_Ext()
   LIN {X -3.161, Y 27.640, Z 85.000}
   LaserEnd_Ext()
   LIN {X -3.411, Y 28.640, Z 85.000}
   LaserStart_Ext()
   LIN {X 4.061, Y 28.640, Z 85.000}
   LaserEnd_Ext()
   LIN {X 3.747, Y 29.640, Z 85.000}
   LaserStart_Ext()
   LIN {X -3.692, Y 29.640, Z 85.000}
   LaserEnd_Ext()
   LIN {X -3.974, Y 30.640, Z 85.000}
   LaserStart_Ext()
   LIN {X 3.386, Y 30.640, Z 85.000}
   LaserEnd_Ext()
   LIN {X 2.992, Y 31.640, Z 85.000}
   LaserStart_Ext()
   LIN {X -4.285, Y 31.640, Z 85.000}
   LaserEnd_Ext()
   LIN {X -4.598, Y 32.640, Z 85.000}
   LaserStart_Ext()
   LIN {X 2.595, Y 32.640, Z 85.000}
   LaserEnd_Ext()
   LIN {X 2.166, Y 33.640, Z 85.000}
   LaserStart_Ext()
   LIN {X -4.926, Y 33.640, Z 85.000}
   LaserEnd_Ext()
   LIN {X -5.289, Y 34.640, Z 85.000}
   LaserStart_Ext()
   LIN {X 1.735, Y 34.640, Z 85.000}
   LaserEnd_Ext()
   LIN {X 1.305, Y 35.640, Z 85.000}
   LaserStart_Ext()
   LIN {X -5.650, Y 35.640, Z 85.000}
   LaserEnd_Ext()
   LIN {X -6.036, Y 36.640, Z 85.000}
   LaserStart_Ext()
   LIN {X 0.874, Y 36.640, Z 85.000}
   LaserEnd_Ext()
   LIN {X 0.426, Y 37.640, Z 85.000}
   LaserStart_Ext()
   LIN {X -6.439, Y 37.640, Z 85.000}
   LaserEnd_Ext()
   LIN {X -6.855, Y 38.640, Z 85.000}
   LaserStart_Ext()
   LIN {X -0.045, Y 38.640, Z 85.000}
   LaserEnd_Ext()
   LIN {X -0.522, Y 39.640, Z 85.000}
   LaserStart_Ext()
   LIN {X -7.289, Y 39.640, Z 85.000}
   LaserEnd_Ext()
   LIN {X -7.740, Y 40.640, Z 85.000}
   LaserStart_Ext()
   LIN {X -1.020, Y 40.640, Z 85.000}
   LaserEnd_Ext()
   LIN {X -1.525, Y 41.640, Z 85.000}
   LaserStart_Ext()
   LIN {X -8.041, Y 41.640, Z 85.000}
   LaserEnd_Ext()
   LIN {X -8.063, Y 42.640, Z 85.000}
   LaserStart_Ext()
   LIN {X -2.039, Y 42.640, Z 85.000}
   LaserEnd_Ext()
   LIN {X -2.607, Y 43.640, Z 85.000}
   LaserStart_Ext()
   LIN {X -7.690, Y 43.640, Z 85.000}
   LaserEnd_Ext()
   LIN {X -6.391, Y 44.640, Z 85.000}
   LaserStart_Ext()
   LIN {X -3.654, Y 44.640, Z 85.000}
   LaserEnd_Ext()
   LIN {X 4.545, Y -14.645, Z 85.850}
   LaserStart_Ext()
   LIN {X 5.280, Y -15.015, Z 85.850} C_DIS
   LIN {X 5.995, Y -15.996, Z 85.850} C_DIS
   LIN {X 6.775, Y -17.072, Z 85.850} C_DIS
   LIN {X 6.933, Y -18.163, Z 85.850} C_DIS
   LIN {X 7.094, Y -19.259, Z 85.850} C_DIS
   LIN {X 6.793, Y -20.219, Z 85.850} C_DIS
   LIN {X 6.408, Y -21.428, Z 85.850} C_DIS
   LIN {X 5.201, Y -22.724, Z 85.850} C_DIS
   LIN {X 4.919, Y -23.028, Z 85.850} C_DIS
   LIN {X 4.687, Y -23.123, Z 85.850} C_DIS
   LIN {X 2.887, Y -23.844, Z 85.850} C_DIS
   LIN {X 1.287, Y -23.779, Z 85.850} C_DIS
   LIN {X 0.810, Y -23.757, Z 85.850} C_DIS
   LIN {X 0.213, Y -23.456, Z 85.850} C_DIS
   LIN {X -1.036, Y -22.828, Z 85.850} C_DIS
   LIN {X -1.715, Y -22.005, Z 85.850} C_DIS
   LIN {X -2.358, Y -21.219, Z 85.850} C_DIS
   LIN {X -2.639, Y -20.161, Z 85.850} C_DIS
   LIN {X -2.896, Y -19.203, Z 85.850} C_DIS
   LIN {X -2.401, Y -17.157, Z 85.850} C_DIS
   LIN {X -2.217, Y -16.408, Z 85.850} C_DIS
   LIN {X -2.017, Y -16.186, Z 85.850} C_DIS
   LIN {X -0.915, Y -14.931, Z 85.850} C_DIS
   LIN {X 0.946, Y -14.126, Z 85.850} C_DIS
   LIN {X 1.296, Y -13.972, Z 85.850} C_DIS
   LIN {X 3.385, Y -14.053, Z 85.850} C_DIS
   LIN {X 4.545, Y -14.645, Z 85.850}
   LaserEnd_Ext()
   LIN {X -3.201, Y 22.985, Z 85.850}
   LaserStart_Ext()
   LIN {X -4.327, Y 28.161, Z 85.850} C_DIS
   LIN {X -4.781, Y 29.775, Z 85.850} C_DIS
   LIN {X -4.941, Y 30.288, Z 85.850} C_DIS
   LIN {X -5.281, Y 31.376, Z 85.850} C_DIS
   LIN {X -5.821, Y 33.097, Z 85.850} C_DIS
   LIN {X -6.409, Y 34.714, Z 85.850} C_DIS
   LIN {X -6.779, Y 35.722, Z 85.850} C_DIS
   LIN {X -7.209, Y 36.779, Z 85.850} C_DIS
   LIN {X -7.671, Y 37.919, Z 85.850} C_DIS
   LIN {X -8.024, Y 38.730, Z 85.850} C_DIS
   LIN {X -8.312, Y 39.384, Z 85.850} C_DIS
   LIN {X -8.589, Y 39.991, Z 85.850} C_DIS
   LIN {X -8.830, Y 40.522, Z 85.850} C_DIS
   LIN {X -8.941, Y 40.941, Z 85.850} C_DIS
   LIN {X -9.198, Y 41.834, Z 85.850} C_DIS
   LIN {X -9.121, Y 42.897, Z 85.850} C_DIS
   LIN {X -9.082, Y 43.273, Z 85.850} C_DIS
   LIN {X -8.853, Y 43.710, Z 85.850} C_DIS
   LIN {X -8.303, Y 44.770, Z 85.850} C_DIS
   LIN {X -6.726, Y 45.681, Z 85.850} C_DIS
   LIN {X -5.922, Y 46.148, Z 85.850} C_DIS
   LIN {X -5.061, Y 46.103, Z 85.850} C_DIS
   LIN {X -4.180, Y 46.059, Z 85.850} C_DIS
   LIN {X -3.707, Y 45.808, Z 85.850} C_DIS
   LIN {X -2.645, Y 45.241, Z 85.850} C_DIS
   LIN {X -1.842, Y 44.246, Z 85.850} C_DIS
   LIN {X -1.721, Y 44.097, Z 85.850} C_DIS
   LIN {X -1.647, Y 43.958, Z 85.850} C_DIS
   LIN {X -1.020, Y 42.779, Z 85.850} C_DIS
   LIN {X -0.207, Y 41.186, Z 85.850} C_DIS
   LIN {X 0.077, Y 40.624, Z 85.850} C_DIS
   LIN {X 1.176, Y 38.336, Z 85.850} C_DIS
   LIN {X 1.486, Y 37.678, Z 85.850} C_DIS
   LIN {X 2.304, Y 35.779, Z 85.850} C_DIS
   LIN {X 3.368, Y 33.335, Z 85.850} C_DIS
   LIN {X 3.754, Y 32.384, Z 85.850} C_DIS
   LIN {X 4.194, Y 31.274, Z 85.850} C_DIS
   LIN {X 4.240, Y 31.161, Z 85.850} C_DIS
   LIN {X 4.591, Y 30.251, Z 85.850} C_DIS
   LIN {X 5.300, Y 27.987, Z 85.850} C_DIS
   LIN {X 7.378, Y 21.810, Z 85.850} C_DIS
   LIN {X 8.729, Y 16.094, Z 85.850} C_DIS
   LIN {X 9.540, Y 12.912, Z 85.850} C_DIS
   LIN {X 10.048, Y 9.680, Z 85.850} C_DIS
   LIN {X 11.163, Y 1.670, Z 85.850} C_DIS
   LIN {X 11.380, Y -2.455, Z 85.850} C_DIS
   LIN {X 11.565, Y -4.760, Z 85.850} C_DIS
   LIN {X 11.581, Y -4.957, Z 85.850} C_DIS
   LIN {X 11.588, Y -5.319, Z 85.850} C_DIS
   LIN {X 11.635, Y -9.744, Z 85.850} C_DIS
   LIN {X 11.591, Y -11.561, Z 85.850} C_DIS
   LIN {X 11.529, Y -13.547, Z 85.850} C_DIS
   LIN {X 11.431, Y -15.139, Z 85.850} C_DIS
   LIN {X 11.356, Y -16.502, Z 85.850} C_DIS
   LIN {X 11.224, Y -18.101, Z 85.850} C_DIS
   LIN {X 11.078, Y -19.753, Z 85.850} C_DIS
   LIN {X 10.313, Y -22.044, Z 85.850} C_DIS
   LIN {X 9.852, Y -23.457, Z 85.850} C_DIS
   LIN {X 9.357, Y -24.036, Z 85.850} C_DIS
   LIN {X 7.881, Y -25.783, Z 85.850} C_DIS
   LIN {X 5.361, Y -27.291, Z 85.850} C_DIS
   LIN {X 2.357, Y -27.915, Z 85.850} C_DIS
   LIN {X -0.288, Y -27.322, Z 85.850} C_DIS
   LIN {X -2.218, Y -26.853, Z 85.850} C_DIS
   LIN {X -3.384, Y -25.952, Z 85.850} C_DIS
   LIN {X -4.566, Y -25.026, Z 85.850} C_DIS
   LIN {X -5.902, Y -22.975, Z 85.850} C_DIS
   LIN {X -6.157, Y -22.586, Z 85.850} C_DIS
   LIN {X -6.264, Y -22.082, Z 85.850} C_DIS
   LIN {X -6.914, Y -18.954, Z 85.850} C_DIS
   LIN {X -6.615, Y -17.323, Z 85.850} C_DIS
   LIN {X -6.352, Y -15.834, Z 85.850} C_DIS
   LIN {X -5.541, Y -13.433, Z 85.850} C_DIS
   LIN {X -5.145, Y -12.283, Z 85.850} C_DIS
   LIN {X -4.866, Y -11.338, Z 85.850} C_DIS
   LIN {X -4.308, Y -9.391, Z 85.850} C_DIS
   LIN {X -3.866, Y -7.538, Z 85.850} C_DIS
   LIN {X -3.460, Y -5.864, Z 85.850} C_DIS
   LIN {X -2.928, Y -3.087, Z 85.850} C_DIS
   LIN {X -2.879, Y -2.834, Z 85.850} C_DIS
   LIN {X -2.450, Y -0.025, Z 85.850} C_DIS
   LIN {X -2.130, Y 3.284, Z 85.850} C_DIS
   LIN {X -1.900, Y 7.012, Z 85.850} C_DIS
   LIN {X -1.908, Y 11.184, Z 85.850} C_DIS
   LIN {X -2.789, Y 20.865, Z 85.850} C_DIS
   LIN {X -2.907, Y 21.683, Z 85.850} C_DIS
   LIN {X -3.201, Y 22.985, Z 85.850}
   LaserEnd_Ext()
   LIN {X 10.602, Y -6.658, Z 85.850}
   LaserStart_Ext()
   LIN {X 10.602, Y -11.095, Z 85.850}
   LaserEnd_Ext()
   LIN {X 9.602, Y -21.015, Z 85.850}
   LaserStart_Ext()
   LIN {X 9.602, Y 5.630, Z 85.850}
   LaserEnd_Ext()
   LIN {X 8.602, Y 12.442, Z 85.850}
   LaserStart_Ext()
   LIN {X 8.602, Y -23.380, Z 85.850}
   LaserEnd_Ext()
   LIN {X 7.602, Y -24.564, Z 85.850}
   LaserStart_Ext()
   LIN {X 7.602, Y -20.974, Z 85.850}
   LaserEnd_Ext()
   LIN {X 7.602, Y -16.511, Z 85.850}
   LaserStart_Ext()
   LIN {X 7.602, Y 16.516, Z 85.850}
   LaserEnd_Ext()
   LIN {X 6.602, Y 20.746, Z 85.850}
   LaserStart_Ext()
   LIN {X 6.602, Y -15.131, Z 85.850}
   LaserEnd_Ext()
   LIN {X 6.602, Y -22.687, Z 85.850}
   LaserStart_Ext()
   LIN {X 6.602, Y -25.383, Z 85.850}
   LaserEnd_Ext()
   LIN {X 5.602, Y -25.981, Z 85.850}
   LaserStart_Ext()
   LIN {X 5.602, Y -23.757, Z 85.850}
   LaserEnd_Ext()
   LIN {X 5.602, Y -14.058, Z 85.850}
   LaserStart_Ext()
   LIN {X 5.602, Y 23.954, Z 85.850}
   LaserEnd_Ext()
   LIN {X 4.602, Y 26.927, Z 85.850}
   LaserStart_Ext()
   LIN {X 4.602, Y -13.551, Z 85.850}
   LaserEnd_Ext()
   LIN {X 4.602, Y -24.234, Z 85.850}
   LaserStart_Ext()
   LIN {X 4.602, Y -26.427, Z 85.850}
   LaserEnd_Ext()
   LIN {X 3.602, Y -26.635, Z 85.850}
   LaserStart_Ext()
   LIN {X 3.602, Y -24.635, Z 85.850}
   LaserEnd_Ext()
   LIN {X 3.602, Y -13.078, Z 85.850}
   LaserStart_Ext()
   LIN {X 3.602, Y 30.038, Z 85.850}
   LaserEnd_Ext()
   LIN {X 2.602, Y 32.564, Z 85.850}
   LaserStart_Ext()
   LIN {X 2.602, Y -13.022, Z 85.850}
   LaserEnd_Ext()
   LIN {X 2.602, Y -24.833, Z 85.850}
   LaserStart_Ext()
   LIN {X 2.602, Y -26.843, Z 85.850}
   LaserEnd_Ext()
   LIN {X 1.602, Y -26.721, Z 85.850}
   LaserStart_Ext()
   LIN {X 1.602, Y -24.792, Z 85.850}
   LaserEnd_Ext()
   LIN {X 1.602, Y -12.983, Z 85.850}
   LaserStart_Ext()
   LIN {X 1.602, Y 34.887, Z 85.850}
   LaserEnd_Ext()
   LIN {X 0.602, Y 37.202, Z 85.850}
   LaserStart_Ext()
   LIN {X 0.602, Y -13.185, Z 85.850}
   LaserEnd_Ext()
   LIN {X 0.602, Y -24.734, Z 85.850}
   LaserStart_Ext()
   LIN {X 0.602, Y -26.497, Z 85.850}
   LaserEnd_Ext()
   LIN {X -0.398, Y -26.266, Z 85.850}
   LaserStart_Ext()
   LIN {X -0.398, Y -24.268, Z 85.850}
   LaserEnd_Ext()
   LIN {X -0.398, Y -13.618, Z 85.850}
   LaserStart_Ext()
   LIN {X -0.398, Y 39.304, Z 85.850}
   LaserEnd_Ext()
   LIN {X -1.398, Y 41.320, Z 85.850}
   LaserStart_Ext()
   LIN {X -1.398, Y 16.615, Z 85.850}
   LaserEnd_Ext()
   LIN {X -1.398, Y 0.460, Z 85.850}
   LaserStart_Ext()
   LIN {X -1.398, Y -14.056, Z 85.850}
   LaserEnd_Ext()
   LIN {X -1.398, Y -23.766, Z 85.850}
   LaserStart_Ext()
   LIN {X -1.398, Y -26.023, Z 85.850}
   LaserEnd_Ext()
   LIN {X -2.398, Y -25.450, Z 85.850}
   LaserStart_Ext()
   LIN {X -2.398, Y -22.749, Z 85.850}
   LaserEnd_Ext()
   LIN {X -2.398, Y -15.104, Z 85.850}
   LaserStart_Ext()
   LIN {X -2.398, Y -5.638, Z 85.850}
   LaserEnd_Ext()
   LIN {X -2.398, Y 23.998, Z 85.850}
   LaserStart_Ext()
   LIN {X -2.398, Y 43.240, Z 85.850}
   LaserEnd_Ext()
   LIN {X -3.398, Y 44.510, Z 85.850}
   LaserStart_Ext()
   LIN {X -3.398, Y 28.552, Z 85.850}
   LaserEnd_Ext()
   LIN {X -3.398, Y -9.846, Z 85.850}
   LaserStart_Ext()
   LIN {X -3.398, Y -17.025, Z 85.850}
   LaserEnd_Ext()
   LIN {X -3.398, Y -21.200, Z 85.850}
   LaserStart_Ext()
   LIN {X -3.398, Y -24.671, Z 85.850}
   LaserEnd_Ext()
   LIN {X -4.398, Y -23.451, Z 85.850}
   LaserStart_Ext()
   LIN {X -4.398, Y -13.185, Z 85.850}
   LaserEnd_Ext()
   LIN {X -4.398, Y 31.901, Z 85.850}
   LaserStart_Ext()
   LIN {X -4.398, Y 45.043, Z 85.850}
   LaserEnd_Ext()
   LIN {X -5.398, Y 45.120, Z 85.850}
   LaserStart_Ext()
   LIN {X -5.398, Y 34.860, Z 85.850}
   LaserEnd_Ext()
   LIN {X -5.398, Y -16.185, Z 85.850}
   LaserStart_Ext()
   LIN {X -5.398, Y -21.335, Z 85.850}
   LaserEnd_Ext()
   LIN {X -6.398, Y 37.440, Z 85.850}
   LaserStart_Ext()
   LIN {X -6.398, Y 44.716, Z 85.850}
   LaserEnd_Ext()
   LIN {X -7.398, Y 44.138, Z 85.850}
   LaserStart_Ext()
   LIN {X -7.398, Y 39.790, Z 85.850}
   LaserEnd_Ext()
   LIN {X 6.851, Y -17.004, Z 86.700}
   LaserStart_Ext()
   LIN {X 6.924, Y -17.486, Z 86.700} C_DIS
   LIN {X 7.175, Y -19.190, Z 86.700} C_DIS
   LIN {X 6.572, Y -21.113, Z 86.700} C_DIS
   LIN {X 6.495, Y -21.360, Z 86.700} C_DIS
   LIN {X 6.370, Y -21.496, Z 86.700} C_DIS
   LIN {X 5.012, Y -22.964, Z 86.700} C_DIS
   LIN {X 3.617, Y -23.530, Z 86.700} C_DIS
   LIN {X 2.979, Y -23.786, Z 86.700} C_DIS
   LIN {X 2.002, Y -23.746, Z 86.700} C_DIS
   LIN {X 0.902, Y -23.704, Z 86.700} C_DIS
   LIN {X 0.211, Y -23.361, Z 86.700} C_DIS
   LIN {X -0.947, Y -22.779, Z 86.700} C_DIS
   LIN {X -2.023, Y -21.474, Z 86.700} C_DIS
   LIN {X -2.273, Y -21.173, Z 86.700} C_DIS
   LIN {X -2.367, Y -20.826, Z 86.700} C_DIS
   LIN {X -2.815, Y -19.158, Z 86.700} C_DIS
   LIN {X -2.406, Y -17.467, Z 86.700} C_DIS
   LIN {X -2.161, Y -16.394, Z 86.700} C_DIS
   LIN {X -1.354, Y -15.449, Z 86.700} C_DIS
   LIN {X -0.881, Y -14.910, Z 86.700} C_DIS
   LIN {X -0.319, Y -14.667, Z 86.700} C_DIS
   LIN {X 1.384, Y -13.914, Z 86.700} C_DIS
   LIN {X 3.419, Y -13.992, Z 86.700} C_DIS
   LIN {X 5.351, Y -14.952, Z 86.700} C_DIS
   LIN {X 6.504, Y -16.532, Z 86.700} C_DIS
   LIN {X 6.851, Y -17.004, Z 86.700}
   LaserEnd_Ext()
   LIN {X 11.563, Y -14.029, Z 86.700}
   LaserStart_Ext()
   LIN {X 11.431, Y -16.424, Z 86.700} C_DIS
   LIN {X 11.200, Y -19.232, Z 86.700} C_DIS
   LIN {X 11.160, Y -19.676, Z 86.700} C_DIS
   LIN {X 10.955, Y -20.291, Z 86.700} C_DIS
   LIN {X 9.953, Y -23.367, Z 86.700} C_DIS
   LIN {X 8.875, Y -24.626, Z 86.700} C_DIS
   LIN {X 7.903, Y -25.776, Z 86.700} C_DIS
   LIN {X 6.239, Y -26.771, Z 86.700} C_DIS
   LIN {X 5.261, Y -27.298, Z 86.700} C_DIS
   LIN {X 3.507, Y -27.617, Z 86.700} C_DIS
   LIN {X 2.314, Y -27.864, Z 86.700} C_DIS
   LIN {X 1.264, Y -27.629, Z 86.700} C_DIS
   LIN {X -2.118, Y -26.807, Z 86.700} C_DIS
   LIN {X -4.164, Y -25.226, Z 86.700} C_DIS
   LIN {X -4.471, Y -24.986, Z 86.700} C_DIS
   LIN {X -4.818, Y -24.453, Z 86.700} C_DIS
   LIN {X -6.068, Y -22.549, Z 86.700} C_DIS
   LIN {X -6.592, Y -20.081, Z 86.700} C_DIS
   LIN {X -6.834, Y -18.919, Z 86.700} C_DIS
   LIN {X -6.723, Y -18.313, Z 86.700} C_DIS
   LIN {X -6.278, Y -15.797, Z 86.700} C_DIS
   LIN {X -5.165, Y -12.498, Z 86.700} C_DIS
   LIN {X -5.068, Y -12.208, Z 86.700} C_DIS
   LIN {X -4.943, Y -11.768, Z 86.700} C_DIS
   LIN {X -4.242, Y -9.321, Z 86.700} C_DIS
   LIN {X -3.528, Y -6.327, Z 86.700} C_DIS
   LIN {X -3.448, Y -5.995, Z 86.700} C_DIS
   LIN {X -3.342, Y -5.443, Z 86.700} C_DIS
   LIN {X -2.865, Y -2.964, Z 86.700} C_DIS
   LIN {X -2.751, Y -2.213, Z 86.700} C_DIS
   LIN {X -2.443, Y -0.200, Z 86.700} C_DIS
   LIN {X -2.084, Y 3.511, Z 86.700} C_DIS
   LIN {X -1.897, Y 6.550, Z 86.700} C_DIS
   LIN {X -1.907, Y 11.533, Z 86.700} C_DIS
   LIN {X -2.640, Y 19.591, Z 86.700} C_DIS
   LIN {X -3.000, Y 22.082, Z 86.700} C_DIS
   LIN {X -3.895, Y 26.041, Z 86.700} C_DIS
   LIN {X -4.414, Y 28.430, Z 86.700} C_DIS
   LIN {X -4.624, Y 29.175, Z 86.700} C_DIS
   LIN {X -4.698, Y 29.412, Z 86.700} C_DIS
   LIN {X -4.855, Y 29.914, Z 86.700} C_DIS
   LIN {X -5.516, Y 32.023, Z 86.700} C_DIS
   LIN {X -5.872, Y 33.160, Z 86.700} C_DIS
   LIN {X -6.226, Y 34.118, Z 86.700} C_DIS
   LIN {X -6.828, Y 35.757, Z 86.700} C_DIS
   LIN {X -7.265, Y 36.832, Z 86.700} C_DIS
   LIN {X -7.724, Y 37.952, Z 86.700} C_DIS
   LIN {X -8.146, Y 38.907, Z 86.700} C_DIS
   LIN {X -8.369, Y 39.415, Z 86.700} C_DIS
   LIN {X -8.521, Y 39.750, Z 86.700} C_DIS
   LIN {X -8.889, Y 40.552, Z 86.700} C_DIS
   LIN {X -9.210, Y 41.606, Z 86.700} C_DIS
   LIN {X -9.248, Y 41.737, Z 86.700} C_DIS
   LIN {X -9.237, Y 41.882, Z 86.700} C_DIS
   LIN {X -9.147, Y 43.308, Z 86.700} C_DIS
   LIN {X -8.370, Y 44.792, Z 86.700} C_DIS
   LIN {X -8.294, Y 44.860, Z 86.700} C_DIS
   LIN {X -5.995, Y 46.185, Z 86.700} C_DIS
   LIN {X -5.110, Y 46.143, Z 86.700} C_DIS
   LIN {X -4.252, Y 46.100, Z 86.700} C_DIS
   LIN {X -3.054, Y 45.464, Z 86.700} C_DIS
   LIN {X -2.716, Y 45.286, Z 86.700} C_DIS
   LIN {X -2.567, Y 45.103, Z 86.700} C_DIS
   LIN {X -1.789, Y 44.143, Z 86.700} C_DIS
   LIN {X -1.118, Y 42.888, Z 86.700} C_DIS
   LIN {X -1.023, Y 42.705, Z 86.700} C_DIS
   LIN {X -0.085, Y 40.878, Z 86.700} C_DIS
   LIN {X 0.215, Y 40.275, Z 86.700} C_DIS
   LIN {X 1.371, Y 37.862, Z 86.700} C_DIS
   LIN {X 1.602, Y 37.360, Z 86.700} C_DIS
   LIN {X 3.191, Y 33.710, Z 86.700} C_DIS
   LIN {X 4.055, Y 31.577, Z 86.700} C_DIS
   LIN {X 4.336, Y 30.870, Z 86.700} C_DIS
   LIN {X 4.384, Y 30.753, Z 86.700} C_DIS
   LIN {X 4.589, Y 30.219, Z 86.700} C_DIS
   LIN {X 5.040, Y 28.777, Z 86.700} C_DIS
   LIN {X 7.373, Y 21.840, Z 86.700} C_DIS
   LIN {X 8.540, Y 16.907, Z 86.700} C_DIS
   LIN {X 9.580, Y 12.826, Z 86.700} C_DIS
   LIN {X 10.230, Y 8.681, Z 86.700} C_DIS
   LIN {X 11.193, Y 1.765, Z 86.700} C_DIS
   LIN {X 11.380, Y -1.797, Z 86.700} C_DIS
   LIN {X 11.541, Y -3.788, Z 86.700} C_DIS
   LIN {X 11.629, Y -4.878, Z 86.700} C_DIS
   LIN {X 11.664, Y -6.887, Z 86.700} C_DIS
   LIN {X 11.694, Y -9.665, Z 86.700} C_DIS
   LIN {X 11.619, Y -12.769, Z 86.700} C_DIS
   LIN {X 11.597, Y -13.468, Z 86.700} C_DIS
   LIN {X 11.563, Y -14.029, Z 86.700}
   LaserEnd_Ext()
   LIN {X -3.411, Y 44.522, Z 86.700}
   LaserStart_Ext()
   LIN {X -6.878, Y 44.522, Z 86.700}
   LaserEnd_Ext()
   LIN {X -7.906, Y 43.522, Z 86.700}
   LaserStart_Ext()
   LIN {X -2.591, Y 43.522, Z 86.700}
   LaserEnd_Ext()
   LIN {X -2.056, Y 42.522, Z 86.700}
   LaserStart_Ext()
   LIN {X -8.195, Y 42.522, Z 86.700}
   LaserEnd_Ext()
   LIN {X -8.139, Y 41.522, Z 86.700}
   LaserStart_Ext()
   LIN {X -1.540, Y 41.522, Z 86.700}
   LaserEnd_Ext()
   LIN {X -1.026, Y 40.522, Z 86.700}
   LaserStart_Ext()
   LIN {X -7.775, Y 40.522, Z 86.700}
   LaserEnd_Ext()
   LIN {X -7.323, Y 39.522, Z 86.700}
   LaserStart_Ext()
   LIN {X -0.533, Y 39.522, Z 86.700}
   LaserEnd_Ext()
   LIN {X -0.054, Y 38.522, Z 86.700}
   LaserStart_Ext()
   LIN {X -6.883, Y 38.522, Z 86.700}
   LaserEnd_Ext()
   LIN {X -6.467, Y 37.522, Z 86.700}
   LaserStart_Ext()
   LIN {X 0.425, Y 37.522, Z 86.700}
   LaserEnd_Ext()
   LIN {X 0.876, Y 36.522, Z 86.700}
   LaserStart_Ext()
   LIN {X -6.059, Y 36.522, Z 86.700}
   LaserEnd_Ext()
   LIN {X -5.676, Y 35.522, Z 86.700}
   LaserStart_Ext()
   LIN {X 1.312, Y 35.522, Z 86.700}
   LaserEnd_Ext()
   LIN {X 1.747, Y 34.522, Z 86.700}
   LaserStart_Ext()
   LIN {X -5.309, Y 34.522, Z 86.700}
   LaserEnd_Ext()
   LIN {X -4.939, Y 33.522, Z 86.700}
   LaserStart_Ext()
   LIN {X 2.183, Y 33.522, Z 86.700}
   LaserEnd_Ext()
   LIN {X 2.594, Y 32.522, Z 86.700}
   LaserStart_Ext()
   LIN {X -4.624, Y 32.522, Z 86.700}
   LaserEnd_Ext()
   LIN {X -4.311, Y 31.522, Z 86.700}
   LaserStart_Ext()
   LIN {X 2.999, Y 31.522, Z 86.700}
   LaserEnd_Ext()
   LIN {X 3.398, Y 30.522, Z 86.700}
   LaserStart_Ext()
   LIN {X -3.997, Y 30.522, Z 86.700}
   LaserEnd_Ext()
   LIN {X -3.685, Y 29.522, Z 86.700}
   LaserStart_Ext()
   LIN {X 3.759, Y 29.522, Z 86.700}
   LaserEnd_Ext()
   LIN {X 4.072, Y 28.522, Z 86.700}
   LaserStart_Ext()
   LIN {X -3.411, Y 28.522, Z 86.700}
   LaserEnd_Ext()
   LIN {X -3.193, Y 27.522, Z 86.700}
   LaserStart_Ext()
   LIN {X 4.408, Y 27.522, Z 86.700}
   LaserEnd_Ext()
   LIN {X 4.744, Y 26.522, Z 86.700}
   LaserStart_Ext()
   LIN {X -2.976, Y 26.522, Z 86.700}
   LaserEnd_Ext()
   LIN {X -2.752, Y 25.522, Z 86.700}
   LaserStart_Ext()
   LIN {X 5.080, Y 25.522, Z 86.700}
   LaserEnd_Ext()
   LIN {X 5.416, Y 24.522, Z 86.700}
   LaserStart_Ext()
   LIN {X -2.526, Y 24.522, Z 86.700}
   LaserEnd_Ext()
   LIN {X -2.300, Y 23.522, Z 86.700}
   LaserStart_Ext()
   LIN {X 5.753, Y 23.522, Z 86.700}
   LaserEnd_Ext()
   LIN {X 6.089, Y 22.522, Z 86.700}
   LaserStart_Ext()
   LIN {X -2.074, Y 22.522, Z 86.700}
   LaserEnd_Ext()
   LIN {X -1.908, Y 21.522, Z 86.700}
   LaserStart_Ext()
   LIN {X 6.421, Y 21.522, Z 86.700}
   LaserEnd_Ext()
   LIN {X 6.658, Y 20.522, Z 86.700}
   LaserStart_Ext()
   LIN {X -1.764, Y 20.522, Z 86.700}
   LaserEnd_Ext()
   LIN {X -1.630, Y 19.522, Z 86.700}
   LaserStart_Ext()
   LIN {X 6.894, Y 19.522, Z 86.700}
   LaserEnd_Ext()
   LIN {X 7.130, Y 18.522, Z 86.700}
   LaserStart_Ext()
   LIN {X -1.539, Y 18.522, Z 86.700}
   LaserEnd_Ext()
   LIN {X -1.448, Y 17.522, Z 86.700}
   LaserStart_Ext()
   LIN {X 7.367, Y 17.522, Z 86.700}
   LaserEnd_Ext()
   LIN {X 7.606, Y 16.522, Z 86.700}
   LaserStart_Ext()
   LIN {X -1.357, Y 16.522, Z 86.700}
   LaserEnd_Ext()
   LIN {X -1.266, Y 15.522, Z 86.700}
   LaserStart_Ext()
   LIN {X 7.861, Y 15.522, Z 86.700}
   LaserEnd_Ext()
   LIN {X 8.116, Y 14.522, Z 86.700}
   LaserStart_Ext()
   LIN {X -1.175, Y 14.522, Z 86.700}
   LaserEnd_Ext()
   LIN {X -1.084, Y 13.522, Z 86.700}
   LaserStart_Ext()
   LIN {X 8.371, Y 13.522, Z 86.700}
   LaserEnd_Ext()
   LIN {X 8.615, Y 12.522, Z 86.700}
   LaserStart_Ext()
   LIN {X -0.993, Y 12.522, Z 86.700}
   LaserEnd_Ext()
   LIN {X -0.907, Y 11.522, Z 86.700}
   LaserStart_Ext()
   LIN {X 8.772, Y 11.522, Z 86.700}
   LaserEnd_Ext()
   LIN {X 8.929, Y 10.522, Z 86.700}
   LaserStart_Ext()
   LIN {X -0.905, Y 10.522, Z 86.700}
   LaserEnd_Ext()
   LIN {X -0.903, Y 9.522, Z 86.700}
   LaserStart_Ext()
   LIN {X 9.086, Y 9.522, Z 86.700}
   LaserEnd_Ext()
   LIN {X 9.243, Y 8.522, Z 86.700}
   LaserStart_Ext()
   LIN {X -0.901, Y 8.522, Z 86.700}
   LaserEnd_Ext()
   LIN {X -0.899, Y 7.522, Z 86.700}
   LaserStart_Ext()
   LIN {X 9.382, Y 7.522, Z 86.700}
   LaserEnd_Ext()
   LIN {X 9.521, Y 6.522, Z 86.700}
   LaserStart_Ext()
   LIN {X -0.898, Y 6.522, Z 86.700}
   LaserEnd_Ext()
   LIN {X -0.958, Y 5.522, Z 86.700}
   LaserStart_Ext()
   LIN {X 9.661, Y 5.522, Z 86.700}
   LaserEnd_Ext()
   LIN {X 9.800, Y 4.522, Z 86.700}
   LaserStart_Ext()
   LIN {X -1.020, Y 4.522, Z 86.700}
   LaserEnd_Ext()
   LIN {X -1.082, Y 3.522, Z 86.700}
   LaserStart_Ext()
   LIN {X 9.939, Y 3.522, Z 86.700}
   LaserEnd_Ext()
   LIN {X 10.078, Y 2.522, Z 86.700}
   LaserStart_Ext()
   LIN {X -1.175, Y 2.522, Z 86.700}
   LaserEnd_Ext()
   LIN {X -1.272, Y 1.522, Z 86.700}
   LaserStart_Ext()
   LIN {X 10.205, Y 1.522, Z 86.700}
   LaserEnd_Ext()
   LIN {X 10.257, Y 0.522, Z 86.700}
   LaserStart_Ext()
   LIN {X -1.369, Y 0.522, Z 86.700}
   LaserEnd_Ext()
   LIN {X -1.474, Y -0.478, Z 86.700}
   LaserStart_Ext()
   LIN {X 10.310, Y -0.478, Z 86.700}
   LaserEnd_Ext()
   LIN {X 10.362, Y -1.478, Z 86.700}
   LaserStart_Ext()
   LIN {X -1.627, Y -1.478, Z 86.700}
   LaserEnd_Ext()
   LIN {X -1.780, Y -2.478, Z 86.700}
   LaserStart_Ext()
   LIN {X 10.432, Y -2.478, Z 86.700}
   LaserEnd_Ext()
   LIN {X 10.513, Y -3.478, Z 86.700}
   LaserStart_Ext()
   LIN {X -1.945, Y -3.478, Z 86.700}
   LaserEnd_Ext()
   LIN {X -2.138, Y -4.478, Z 86.700}
   LaserStart_Ext()
   LIN {X 10.594, Y -4.478, Z 86.700}
   LaserEnd_Ext()
   LIN {X 10.640, Y -5.478, Z 86.700}
   LaserStart_Ext()
   LIN {X -2.330, Y -5.478, Z 86.700}
   LaserEnd_Ext()
   LIN {X -2.536, Y -6.478, Z 86.700}
   LaserStart_Ext()
   LIN {X 10.657, Y -6.478, Z 86.700}
   LaserEnd_Ext()
   LIN {X 10.671, Y -7.478, Z 86.700}
   LaserStart_Ext()
   LIN {X -2.775, Y -7.478, Z 86.700}
   LaserEnd_Ext()
   LIN {X -3.013, Y -8.478, Z 86.700}
   LaserStart_Ext()
   LIN {X 10.681, Y -8.478, Z 86.700}
   LaserEnd_Ext()
   LIN {X 10.692, Y -9.478, Z 86.700}
   LaserStart_Ext()
   LIN {X -3.252, Y -9.478, Z 86.700}
   LaserEnd_Ext()
   LIN {X -3.534, Y -10.478, Z 86.700}
   LaserStart_Ext()
   LIN {X 10.674, Y -10.478, Z 86.700}
   LaserEnd_Ext()
   LIN {X 10.650, Y -11.478, Z 86.700}
   LaserStart_Ext()
   LIN {X -3.820, Y -11.478, Z 86.700}
   LaserEnd_Ext()
   LIN {X -4.105, Y -12.478, Z 86.700}
   LaserStart_Ext()
   LIN {X 10.626, Y -12.478, Z 86.700}
   LaserEnd_Ext()
   LIN {X 10.595, Y -13.478, Z 86.700}
   LaserStart_Ext()
   LIN {X 4.652, Y -13.478, Z 86.700}
   LaserEnd_Ext()
   LIN {X -0.104, Y -13.478, Z 86.700}
   LaserStart_Ext()
   LIN {X -4.440, Y -13.478, Z 86.700}
   LaserEnd_Ext()
   LIN {X -4.778, Y -14.478, Z 86.700}
   LaserStart_Ext()
   LIN {X -1.833, Y -14.478, Z 86.700}
   LaserEnd_Ext()
   LIN {X 6.244, Y -14.478, Z 86.700}
   LaserStart_Ext()
   LIN {X 10.537, Y -14.478, Z 86.700}
   LaserEnd_Ext()
   LIN {X 10.482, Y -15.478, Z 86.700}
   LaserStart_Ext()
   LIN {X 6.973, Y -15.478, Z 86.700}
   LaserEnd_Ext()
   LIN {X -2.694, Y -15.478, Z 86.700}
   LaserStart_Ext()
   LIN {X -5.115, Y -15.478, Z 86.700}
   LaserEnd_Ext()
   LIN {X -5.383, Y -16.478, Z 86.700}
   LaserStart_Ext()
   LIN {X -3.206, Y -16.478, Z 86.700}
   LaserEnd_Ext()
   LIN {X 7.701, Y -16.478, Z 86.700}
   LaserStart_Ext()
   LIN {X 10.424, Y -16.478, Z 86.700}
   LaserEnd_Ext()
   LIN {X 10.341, Y -17.478, Z 86.700}
   LaserStart_Ext()
   LIN {X 7.934, Y -17.478, Z 86.700}
   LaserEnd_Ext()
   LIN {X -3.438, Y -17.478, Z 86.700}
   LaserStart_Ext()
   LIN {X -5.560, Y -17.478, Z 86.700}
   LaserEnd_Ext()
   LIN {X -5.736, Y -18.478, Z 86.700}
   LaserStart_Ext()
   LIN {X -3.679, Y -18.478, Z 86.700}
   LaserEnd_Ext()
   LIN {X 8.081, Y -18.478, Z 86.700}
   LaserStart_Ext()
   LIN {X 10.259, Y -18.478, Z 86.700}
   LaserEnd_Ext()
   LIN {X 10.172, Y -19.478, Z 86.700}
   LaserStart_Ext()
   LIN {X 8.133, Y -19.478, Z 86.700}
   LaserEnd_Ext()
   LIN {X -3.765, Y -19.478, Z 86.700}
   LaserStart_Ext()
   LIN {X -5.696, Y -19.478, Z 86.700}
   LaserEnd_Ext()
   LIN {X -5.486, Y -20.478, Z 86.700}
   LaserStart_Ext()
   LIN {X -3.496, Y -20.478, Z 86.700}
   LaserEnd_Ext()
   LIN {X 7.819, Y -20.478, Z 86.700}
   LaserStart_Ext()
   LIN {X 9.842, Y -20.478, Z 86.700}
   LaserEnd_Ext()
   LIN {X 9.516, Y -21.478, Z 86.700}
   LaserStart_Ext()
   LIN {X 7.505, Y -21.478, Z 86.700}
   LaserEnd_Ext()
   LIN {X -3.224, Y -21.478, Z 86.700}
   LaserStart_Ext()
   LIN {X -5.273, Y -21.478, Z 86.700}
   LaserEnd_Ext()
   LIN {X -4.918, Y -22.478, Z 86.700}
   LaserStart_Ext()
   LIN {X -2.491, Y -22.478, Z 86.700}
   LaserEnd_Ext()
   LIN {X 6.824, Y -22.478, Z 86.700}
   LaserStart_Ext()
   LIN {X 9.191, Y -22.478, Z 86.700}
   LaserEnd_Ext()
   LIN {X 8.541, Y -23.478, Z 86.700}
   LaserStart_Ext()
   LIN {X 5.898, Y -23.478, Z 86.700}
   LaserEnd_Ext()
   LIN {X -1.661, Y -23.478, Z 86.700}
   LaserStart_Ext()
   LIN {X -4.262, Y -23.478, Z 86.700}
   LaserEnd_Ext()
   LIN {X -3.496, Y -24.478, Z 86.700}
   LaserStart_Ext()
   LIN {X 0.214, Y -24.478, Z 86.700}
   LaserEnd_Ext()
   LIN {X 3.940, Y -24.478, Z 86.700}
   LaserStart_Ext()
   LIN {X 7.690, Y -24.478, Z 86.700}
   LaserEnd_Ext()
   LIN {X 6.453, Y -25.478, Z 86.700}
   LaserStart_Ext()
   LIN {X -2.202, Y -25.478, Z 86.700}
   LaserEnd_Ext()
   LIN {X 0.765, Y -26.478, Z 86.700}
   LaserStart_Ext()
   LIN {X 4.178, Y -26.478, Z 86.700}
   LaserEnd_Ext()
   LIN {X 5.422, Y -14.888, Z 87.550}
   LaserStart_Ext()
   LIN {X 5.517, Y -15.018, Z 87.550} C_DIS
   LIN {X 6.928, Y -16.937, Z 87.550} C_DIS
   LIN {X 7.223, Y -18.892, Z 87.550} C_DIS
   LIN {X 7.257, Y -19.122, Z 87.550} C_DIS
   LIN {X 7.175, Y -19.382, Z 87.550} C_DIS
   LIN {X 6.583, Y -21.291, Z 87.550} C_DIS
   LIN {X 5.621, Y -22.340, Z 87.550} C_DIS
   LIN {X 5.104, Y -22.899, Z 87.550} C_DIS
   LIN {X 3.931, Y -23.376, Z 87.550} C_DIS
   LIN {X 3.074, Y -23.727, Z 87.550} C_DIS
   LIN {X 2.510, Y -23.708, Z 87.550} C_DIS
   LIN {X 0.994, Y -23.650, Z 87.550} C_DIS
   LIN {X -0.815, Y -22.751, Z 87.550} C_DIS
   LIN {X -0.896, Y -22.683, Z 87.550} C_DIS
   LIN {X -2.187, Y -21.127, Z 87.550} C_DIS
   LIN {X -2.676, Y -19.330, Z 87.550} C_DIS
   LIN {X -2.734, Y -19.114, Z 87.550} C_DIS
   LIN {X -2.681, Y -18.894, Z 87.550} C_DIS
   LIN {X -2.109, Y -16.389, Z 87.550} C_DIS
   LIN {X -1.262, Y -15.396, Z 87.550} C_DIS
   LIN {X -0.817, Y -14.866, Z 87.550} C_DIS
   LIN {X 0.391, Y -14.334, Z 87.550} C_DIS
   LIN {X 1.472, Y -13.856, Z 87.550} C_DIS
   LIN {X 3.523, Y -13.934, Z 87.550} C_DIS
   LIN {X 5.269, Y -14.811, Z 87.550} C_DIS
   LIN {X 5.422, Y -14.888, Z 87.550}
   LaserEnd_Ext()
   LIN {X -4.325, Y 46.141, Z 87.550}
   LaserStart_Ext()
   LIN {X -3.837, Y 45.885, Z 87.550} C_DIS
   LIN {X -2.787, Y 45.330, Z 87.550} C_DIS
   LIN {X -1.943, Y 44.295, Z 87.550} C_DIS
   LIN {X -1.857, Y 44.190, Z 87.550} C_DIS
   LIN {X -1.806, Y 44.096, Z 87.550} C_DIS
   LIN {X -1.155, Y 42.883, Z 87.550} C_DIS
   LIN {X -0.453, Y 41.532, Z 87.550} C_DIS
   LIN {X -0.248, Y 41.132, Z 87.550} C_DIS
   LIN {X 0.473, Y 39.681, Z 87.550} C_DIS
   LIN {X 1.174, Y 38.219, Z 87.550} C_DIS
   LIN {X 1.935, Y 36.564, Z 87.550} C_DIS
   LIN {X 3.014, Y 34.085, Z 87.550} C_DIS
   LIN {X 4.357, Y 30.770, Z 87.550} C_DIS
   LIN {X 4.478, Y 30.466, Z 87.550} C_DIS
   LIN {X 4.586, Y 30.186, Z 87.550} C_DIS
   LIN {X 4.780, Y 29.567, Z 87.550} C_DIS
   LIN {X 7.369, Y 21.870, Z 87.550} C_DIS
   LIN {X 8.350, Y 17.719, Z 87.550} C_DIS
   LIN {X 9.619, Y 12.740, Z 87.550} C_DIS
   LIN {X 10.413, Y 7.681, Z 87.550} C_DIS
   LIN {X 11.224, Y 1.859, Z 87.550} C_DIS
   LIN {X 11.381, Y -1.139, Z 87.550} C_DIS
   LIN {X 11.517, Y -2.815, Z 87.550} C_DIS
   LIN {X 11.677, Y -4.800, Z 87.550} C_DIS
   LIN {X 11.741, Y -8.455, Z 87.550} C_DIS
   LIN {X 11.753, Y -9.586, Z 87.550} C_DIS
   LIN {X 11.698, Y -11.870, Z 87.550} C_DIS
   LIN {X 11.666, Y -13.390, Z 87.550} C_DIS
   LIN {X 11.637, Y -13.962, Z 87.550} C_DIS
   LIN {X 11.507, Y -16.345, Z 87.550} C_DIS
   LIN {X 11.305, Y -18.786, Z 87.550} C_DIS
   LIN {X 11.243, Y -19.598, Z 87.550} C_DIS
   LIN {X 11.007, Y -20.351, Z 87.550} C_DIS
   LIN {X 10.053, Y -23.276, Z 87.550} C_DIS
   LIN {X 8.392, Y -25.216, Z 87.550} C_DIS
   LIN {X 7.925, Y -25.769, Z 87.550} C_DIS
   LIN {X 7.125, Y -26.248, Z 87.550} C_DIS
   LIN {X 5.164, Y -27.303, Z 87.550} C_DIS
   LIN {X 2.653, Y -27.759, Z 87.550} C_DIS
   LIN {X 2.103, Y -27.772, Z 87.550} C_DIS
   LIN {X 0.860, Y -27.460, Z 87.550} C_DIS
   LIN {X -2.019, Y -26.761, Z 87.550} C_DIS
   LIN {X -3.220, Y -25.833, Z 87.550} C_DIS
   LIN {X -4.376, Y -24.945, Z 87.550} C_DIS
   LIN {X -4.812, Y -24.289, Z 87.550} C_DIS
   LIN {X -5.978, Y -22.512, Z 87.550} C_DIS
   LIN {X -6.604, Y -19.571, Z 87.550} C_DIS
   LIN {X -6.753, Y -18.884, Z 87.550} C_DIS
   LIN {X -6.642, Y -18.235, Z 87.550} C_DIS
   LIN {X -6.205, Y -15.761, Z 87.550} C_DIS
   LIN {X -5.526, Y -13.750, Z 87.550} C_DIS
   LIN {X -5.052, Y -12.331, Z 87.550} C_DIS
   LIN {X -4.442, Y -10.179, Z 87.550} C_DIS
   LIN {X -4.177, Y -9.251, Z 87.550} C_DIS
   LIN {X -3.826, Y -7.782, Z 87.550} C_DIS
   LIN {X -3.434, Y -6.125, Z 87.550} C_DIS
   LIN {X -3.309, Y -5.477, Z 87.550} C_DIS
   LIN {X -2.851, Y -3.095, Z 87.550} C_DIS
   LIN {X -2.635, Y -1.669, Z 87.550} C_DIS
   LIN {X -2.437, Y -0.374, Z 87.550} C_DIS
   LIN {X -2.039, Y 3.739, Z 87.550} C_DIS
   LIN {X -1.894, Y 6.087, Z 87.550} C_DIS
   LIN {X -1.906, Y 11.882, Z 87.550} C_DIS
   LIN {X -2.492, Y 18.318, Z 87.550} C_DIS
   LIN {X -3.093, Y 22.481, Z 87.550} C_DIS
   LIN {X -4.478, Y 28.609, Z 87.550} C_DIS
   LIN {X -4.508, Y 28.713, Z 87.550} C_DIS
   LIN {X -4.749, Y 29.476, Z 87.550} C_DIS
   LIN {X -5.914, Y 33.197, Z 87.550} C_DIS
   LIN {X -6.454, Y 34.659, Z 87.550} C_DIS
   LIN {X -6.876, Y 35.792, Z 87.550} C_DIS
   LIN {X -7.365, Y 36.978, Z 87.550} C_DIS
   LIN {X -7.778, Y 37.984, Z 87.550} C_DIS
   LIN {X -8.018, Y 38.529, Z 87.550} C_DIS
   LIN {X -8.426, Y 39.446, Z 87.550} C_DIS
   LIN {X -8.940, Y 40.564, Z 87.550} C_DIS
